// Adds a generic item at the back of the deque.
METHOD Enqueue_Generic : I_Deque
VAR_INPUT
	Item : T_Generic; // Item to store.
	bAt_Front : BOOL; // Enqueues at front if set to TRUE.
END_VAR
VAR_OUTPUT
	bSuccess : BOOL;
END_VAR
Enqueue_Generic := THIS^;

IF bAt_Front THEN
	THIS^.fbList.Insert_Generic(0, Item, bSuccess => bSuccess);
ELSE
	THIS^.fbList.Insert_Generic(THIS^.fbList._Count, Item, bSuccess => bSuccess);
	END_IF
END_METHOD

// Get item at the front of the deque without removing it.
METHOD Front : I_Deque
VAR_INPUT
	Item : ANY; // Variable to store returned item value
END_VAR
VAR_OUTPUT
	bSuccess : BOOL;
END_VAR
Front := THIS^;

THIS^.fbList.Get(0, Item, bSuccess => bSuccess);
END_METHOD

// Reverses the order of items in the deque.
METHOD Reverse : I_Deque
VAR_OUTPUT
	bSuccess : BOOL;
END_VAR
Reverse := THIS^;

THIS^.fbList.Reverse(bSuccess => bSuccess);
END_METHOD

END_FUNCTION_BLOCK

// POUs/Function Blocks/Collections/FB_List
// A doubly linked list with iterator hint optimisation.
// Essentially the linked list keeps track of the node it last accessed.
// Iteration starts from the closest node (head, tail or last accessed) to the access/mutation index.
// This should result in sequential access times of O(1) and similar times for access/mutation on the same index.
{attribute 'enable_dynamic_creation'}
{attribute 'no_assign'}
{attribute 'no_explicit_call' := 'direct call for this function block is not allowed'}
FUNCTION_BLOCK FB_List EXTENDS FB_Collection IMPLEMENTS I_List, I_Iterable//, I_Enumerable, I_Copyable
VAR
	pHead, pTail, pLast_Accessed : POINTER TO T_List_Node;
	Last_Accessed_Index : T_Position := -1;
END_VAR

// Iteration helper method that finds the closest node to an index and iterates from there to the node at the specified index.
METHOD PROTECTED Closest_Node_Iterator : POINTER TO T_List_Node
VAR_INPUT
	Index : T_Position;
END_VAR
VAR
	pTmp : POINTER TO T_List_Node;
	Dist, Last_Access_Dist,
	Head_Dist, Tail_Dist : T_Position;
END_VAR
Last_Access_Dist := ABS(THIS^.Last_Accessed_Index - Index);
Head_Dist := Index;
Tail_Dist := THIS^._Count - Index - 1;

Dist := MIN(Last_Access_Dist, Head_Dist, Tail_Dist);

Closest_Node_Iterator := THIS^.Iterate(
	SEL(Dist = Head_Dist, SEL(Dist = Tail_Dist,  THIS^.pLast_Accessed, THIS^.pTail), THIS^.pHead), // Select the closest node to start iteration.
	Dist, // get the smallest displacement
	SEL(Dist = Head_Dist, SEL(Dist = Tail_Dist, Index > THIS^.Last_Accessed_Index, FALSE), TRUE)); // Set the iteration direction.
END_METHOD

// Iteration helper method to iterate from a given node in a specific direction for a specified count.
METHOD PROTECTED Iterate : POINTER TO T_List_Node
VAR_INPUT
	pStart 		: POINTER TO T_List_Node;
	Count 		: T_Capacity;
	bIterateUp 	: BOOL;
END_VAR
VAR
	i : T_Capacity;
END_VAR
Iterate := pStart;
IF Count = 0 THEN RETURN; END_IF
IF bIterateUp THEN FOR i := 0 TO Count - 1 DO Iterate := Iterate^.pNext; END_FOR RETURN; END_IF
FOR i := 0 TO Count - 1 DO Iterate := Iterate^.pPrevious; END_FOR
END_METHOD

// Index of the first element.
PROPERTY _Begin : T_Position
GET
_Begin := 0;
END_GET
END_PROPERTY

// Index of the last element.
PROPERTY _End : T_Position
GET
_End := TO_DINT(THIS^._Count) - 1;
END_GET
END_PROPERTY

// Adds an item to the end of the list.
METHOD Append : I_List
VAR_INPUT
	Item : ANY; // Value to store in list
END_VAR
VAR_OUTPUT
	bSuccess : BOOL;
END_VAR
Append := THIS^;

THIS^.Insert_Generic(THIS^._Count, Item, bSuccess => bSuccess);
END_METHOD

// Empties/Clears/Deletes every item in the list.
METHOD Clear : I_List
VAR
	pTmp : POINTER TO T_List_Node;
END_VAR
Clear := THIS^;

WHILE THIS^.pHead <> 0 DO
	pTmp := THIS^.pHead^.pNext;
	F_Delete_Generic(THIS^.pHead^.Data);
	__DELETE(THIS^.pHead);
	THIS^.pHead := pTmp;
	END_WHILE

THIS^._Count := 0;	
THIS^.pTail := THIS^.pLast_Accessed := 0;
THIS^.Last_Accessed_Index := -1;
THIS^.Clear_Error();
END_METHOD

// Checks if item is contained in list.
METHOD Contains : BOOL
VAR_INPUT
	Item : ANY; // Item to find in list
END_VAR
THIS^.Search(Item, bSuccess => Contains);
END_METHOD

{attribute 'hide'}
METHOD FB_exit : BOOL
VAR_INPUT
	bInCopyCode : BOOL; // if TRUE, the exit method is called for exiting an instance that is copied afterwards (online change).
END_VAR
// If this is an online change or this collection is empty then ignore. 
IF bInCopyCode THEN RETURN; END_IF

THIS^.Clear();
END_METHOD

// Gets item from list at specified location without removing it
METHOD Get : I_List
VAR_INPUT
	Index : T_Position; // Location of item
	Item : ANY;  // Variable to store returned item
END_VAR
VAR_OUTPUT
	bSuccess : BOOL;
END_VAR
VAR
	Tmp : T_Generic;
END_VAR
Get := THIS^;

THIS^.Get_Generic(Index, Item => Tmp, bSuccess => bSuccess);

IF NOT bSuccess THEN RETURN; END_IF

IF NOT F_Matching_Generics(Item, Tmp) THEN
	THIS^._Error_Status := GVL_Errors.ERR_TYPE_MISMATCH;
	bSuccess := FALSE;
	RETURN;
	END_IF
	
F_Copy_Generic_Value(Tmp, Item, bSuccess => bSuccess, Error => THIS^.Error);
END_METHOD

// Returns item as a string, if type to string conversion is supported
METHOD Get_As_String : I_List
VAR_INPUT
	Index : T_Position; // Location of item
	sItem : REFERENCE TO STRING; // Variable to store returned item.
END_VAR
VAR_OUTPUT
	bSuccess : BOOL;
END_VAR
VAR
	Tmp : T_Generic;
END_VAR
Get_As_String := THIS^;

IF NOT __ISVALIDREF(sItem) THEN THIS^._Error_Status := GVL_Errors.ERR_INVALID_REFERENCE; RETURN; END_IF
	
THIS^.Get_Generic(Index, Item => Tmp, bSuccess => bSuccess);

IF NOT bSuccess THEN RETURN; END_IF
	
CASE Tmp.TypeClass OF
	T_Type.TYPE_STRING:
		Tc2_Utilities.STRNCPY(ADR(sItem), Tmp.pValue, MIN(Tc2_Utilities.LEN2(ADR(sItem))+1, TO_UDINT(Tmp.diSize)));
		THIS^.Clear_Error();

	T_Type.TYPE_WSTRING:
		Tc2_Utilities.WSTRING_TO_STRING2(ADR(sItem), Tmp.pValue, MIN(Tc2_Utilities.LEN2(ADR(sItem))+1, TO_UDINT(Tmp.diSize)));
		THIS^.Clear_Error();
ELSE
	sItem := F_Generic_To_String(Tmp, bSuccess => bSuccess, Error => THIS^.Error);
	END_CASE
END_METHOD

// Gets a value from a list in it's generic form.
// (** Use carefully as this contains the pointer of the actual value in the collection. **)
// If you wish to use this it is recommeded you create a copy of the returned value using MEMMOVE or MEMCPY
METHOD Get_Generic : I_List
VAR_INPUT
	Index : T_Position; // Location of item
END_VAR
VAR_OUTPUT
	Item : T_Generic := (TypeClass := T_Type.TYPE_NONE);
	bSuccess : BOOL;
END_VAR
VAR
	pTmp : POINTER TO T_List_Node;
END_VAR
Get_Generic := THIS^;

IF Index < 0 OR_ELSE Index >= THIS^._Count THEN
	// Throw out of bounds error.
	THIS^._Error_Status := GVL_Errors.ERR_INDEX_OUT_OF_BOUNDS;
	RETURN;
	END_IF
	
IF Index = 0 THEN
	Item := THIS^.pHead^.Data;
ELSIF Index = THIS^._Count - 1 THEN
	Item := THIS^.pTail^.Data;
ELSIF Index = THIS^.Last_Accessed_Index THEN
	Item := THIS^.pLast_Accessed^.Data;
ELSE
	pTmp := THIS^.Closest_Node_Iterator(Index);
	Item := pTmp^.Data;
	
	THIS^.Last_Accessed_Index := Index;
	THIS^.pLast_Accessed := pTmp;
	
	END_IF
	
bSuccess := TRUE;
THIS^.Clear_Error();
END_METHOD

// Gets the type of the item at specified location.
METHOD Get_Type_At : I_List
VAR_INPUT
	Index : T_Position;
END_VAR
VAR_OUTPUT
	Item_Type : T_Type := T_Type.TYPE_NONE;
	bSuccess : BOOL;
END_VAR
VAR
	Tmp : T_Generic;
END_VAR
Get_Type_At := THIS^;

THIS^.Get_Generic(Index, Item => Tmp, bSuccess => bSuccess);
Item_Type := Tmp.TypeClass;
END_METHOD

// Adds new item to list at specified location, if index = 0, item will be added at the front, if index = count, item will be added at the back
METHOD Insert : I_List
VAR_INPUT
	Index : T_Position; // Location of item
	Item : ANY; // Item to store in list
END_VAR
VAR_OUTPUT
	bSuccess : BOOL;
END_VAR
Insert := THIS^;

THIS^.Insert_Generic(Index, Item, bSuccess => bSuccess);
END_METHOD

// Adds new item to list at specified location using the generic form. 
// If index = 0, item will be added at the front, if index = count, item will be added at the back
METHOD Insert_Generic : I_List
VAR_INPUT
	Index 	 : T_Position; 	// Location of item
	Item 	 : T_Generic;  	// Item to store in list
END_VAR
VAR_OUTPUT
	bSuccess : BOOL;
END_VAR
VAR
	pTmp, pCurrent : POINTER TO ST_LIST_NODE;
END_VAR
Insert_Generic := THIS^;

IF Index < 0 OR_ELSE Index > THIS^._Count THEN
	// Throw out of bounds error.
	THIS^._Error_Status := GVL_Errors.ERR_INDEX_OUT_OF_BOUNDS;
	RETURN;
	END_IF
	
pTmp := __NEW(ST_LIST_NODE);
IF pTmp = 0 THEN THIS^._Error_Status := GVL_Errors.ERR_MALLOC_FAILED; RETURN; END_IF

pTmp^.Data := F_Clone_Generic(Item, bSuccess => bSuccess, Error => THIS^.Error);
IF NOT bSuccess THEN __DELETE(pTmp); RETURN; END_IF

IF Index = 0 THEN
	//...
	pTmp^.pNext := THIS^.pHead;
	IF THIS^.pHead <> 0 THEN THIS^.pHead^.pPrevious := pTmp; END_IF
	IF THIS^.pTail = 0 THEN THIS^.pTail := pTmp; END_IF
	THIS^.pHead := pTmp;
ELSIF Index = THIS^._Count THEN
	//...
	pTmp^.pPrevious := THIS^.pTail;
	IF THIS^.pTail <> 0 THEN THIS^.pTail^.pNext := pTmp; END_IF
	THIS^.pTail := pTmp;
ELSE	
	pCurrent := THIS^.Closest_Node_Iterator(Index);
	
	pTmp^.pNext := pCurrent;
	pTmp^.pPrevious := pCurrent^.pNext;
	pCurrent^.pPrevious^.pNext := pTmp;
	pCurrent^.pPrevious := pTmp;
	
	THIS^.Last_Accessed_Index := Index;
	THIS^.pLast_Accessed := pTmp;
	END_IF
	
THIS^.Increment_Count();
END_METHOD

// Adds an item at the front of the list.
METHOD Prepend : I_List
VAR_INPUT
	Item : ANY; // Value to store in list
END_VAR
VAR_OUTPUT
	bSuccess : BOOL;
END_VAR
Prepend := THIS^;

THIS^.Insert_Generic(0, Item, bSuccess => bSuccess);
END_METHOD

// Removes item from the list.
METHOD Remove : I_List
VAR_INPUT
	Item : ANY; // Item to remove from in list
END_VAR
VAR_OUTPUT
	bSuccess : BOOL;
END_VAR
VAR
	Tmp : T_Position;
END_VAR
Remove := THIS^;

THIS^.Search(Item, Index => Tmp, bSuccess => bSuccess);
IF NOT bSuccess THEN RETURN; END_IF 
THIS^.Remove_At(Tmp, bSuccess => bSuccess);
END_METHOD

// Remove item at specified location 
METHOD Remove_At : I_List
VAR_INPUT
	Index : T_Position; // Location of item
END_VAR
VAR_OUTPUT
	bSuccess : BOOL;
END_VAR
VAR
	pTmp : POINTER TO T_List_Node;
END_VAR
Remove_At := THIS^;

IF Index < 0 OR_ELSE Index >= THIS^._Count THEN
	// Throw out of bounds error.
	THIS^._Error_Status := GVL_Errors.ERR_INDEX_OUT_OF_BOUNDS;
	RETURN;
	END_IF

IF Index = 0 THEN
	//...
	pTmp := THIS^.pHead;
	IF THIS^.pHead = THIS^.pTail THEN
		THIS^.pLast_Accessed := THIS^.pTail := 0;
		THIS^.Last_Accessed_Index := -1;
		END_IF
		
	THIS^.pHead := THIS^.pHead^.pNext;
	
	F_Delete_Generic(pTmp^.Data);
	__DELETE(pTmp);
	
ELSIF Index = THIS^._Count - 1 THEN
	//...
	pTmp := THIS^.pTail^.pPrevious;
	THIS^.pTail := pTmp;
	F_Delete_Generic(pTmp^.pNext^.Data);
	__DELETE(pTmp^.pNext);
ELSE
	//...	
	pTmp := THIS^.Closest_Node_Iterator(Index);
	
	// Do deletion
	pTmp^.pNext^.pPrevious := pTmp^.pPrevious;
	pTmp^.pPrevious^.pNext := pTmp^.pNext;
	
	THIS^.Last_Accessed_Index := -1;
	THIS^.pLast_Accessed := 0;
	
	THIS^.Last_Accessed_Index := Index;
	THIS^.pLast_Accessed := pTmp^.pNext;
	
	F_Delete_Generic(pTmp^.Data);
	__DELETE(pTmp);
	END_IF
	
THIS^.Decrement_Count();
bSuccess := TRUE;
THIS^.Clear_Error();
END_METHOD

// Removes item at the back of the list.
METHOD Remove_Last : I_List
VAR_OUTPUT
	bSuccess : BOOL;
END_VAR
Remove_Last := THIS^.Remove_At(THIS^._Count - 1, bSuccess => bSuccess);
END_METHOD

// Manually resize list. If list becomes smaller, item on higher locations will be deleted.
METHOD Resize : I_List
VAR_INPUT
	Size : T_Capacity; // New size of list.
END_VAR
VAR_OUTPUT
	bSuccess : BOOL;
END_VAR
VAR
	Tmp : T_Generic := (TypeClass := T_Type.TYPE_NONE);
END_VAR
Resize := THIS^;

IF Size = 0 THEN 
	THIS^.Clear();
ELSE
	WHILE THIS^._Count > Size DO 
		THIS^.Remove_At(THIS^._Count - 1, bSuccess => bSuccess);
		IF NOT bSuccess THEN RETURN; END_IF 
		END_WHILE
	WHILE THIS^._Count < Size DO 
		THIS^.Insert_Generic(THIS^._Count, Tmp, bSuccess => bSuccess);
		IF NOT bSuccess THEN RETURN; END_IF 
		END_WHILE
	END_IF
END_METHOD

// Reverses the order of items in the list
METHOD Reverse : I_List
VAR_OUTPUT
	bSuccess : BOOL;
END_VAR
VAR
	pFront, pBack : POINTER TO T_List_Node;
END_VAR
Reverse := THIS^;

IF THIS^._Empty THEN bSuccess := TRUE; THIS^.Clear_Error(); RETURN; END_IF

pFront := THIS^.pHead;
pBack := THIS^.pTail;

WHILE (pFront <> pBack) AND_THEN (pFront^.pPrevious <> pBack) DO
	F_Swap_Generics(pFront^.Data, pBack^.Data);
	pFront := pFront^.pNext;
	pBack := pBack^.pPrevious;
	END_WHILE
	
bSuccess := TRUE;
THIS^.Clear_Error();
END_METHOD

// Find the location of an item in list.
METHOD Search : I_List
VAR_INPUT
	Item : ANY; // Item to find in list
END_VAR
VAR_OUTPUT
	Index : T_Position := -1; //Location of item in list 
	bSuccess : BOOL;
END_VAR
VAR
	i : T_Position;
	pTmp : POINTER TO T_List_Node;
END_VAR
Search := THIS^;

pTmp := THIS^.pHead; 
WHILE pTmp <> 0 DO
	CASE F_Compare_Generics(Item, pTmp^.Data) OF
		T_Comparison.Equal:
			bSuccess := TRUE;
			THIS^.Clear_Error();
			Index := i;
			RETURN;
		END_CASE
	pTmp := pTmp^.pNext;	
	i := i + 1;
	END_WHILE

// Throw item not found error.
THIS^._Error_Status := GVL_Errors.ERR_NO_ITEM;
END_METHOD

// Changes the item at the specified location in the list.
METHOD Set : I_List
VAR_INPUT
	Index 	: T_Position; // Location of item
	Item 	: ANY; 	// Item to store in list
END_VAR
VAR_OUTPUT
	bSuccess : BOOL;
END_VAR
Set := THIS^;

THIS^.Set_Generic(Index, Item, bSuccess => bSuccess);
END_METHOD

// Changes the item at the specified location in the list in it's generic form.
METHOD Set_Generic : I_List
VAR_INPUT
	Index : T_Position; // Location of item
	Item : T_Generic; // Item to store in list
END_VAR
VAR_OUTPUT
	bSuccess : BOOL;
END_VAR
VAR
	pTmp : POINTER TO T_List_Node;
	Tmp : T_Generic;
END_VAR
Set_Generic := THIS^;

IF Index < 0 OR_ELSE Index >= THIS^._Count THEN
	// Throw out of bounds error.
	THIS^._Error_Status := GVL_Errors.ERR_INDEX_OUT_OF_BOUNDS;
	RETURN;
	END_IF
	
IF Index = 0 THEN
	Tmp := F_Clone_Generic(Item, bSuccess => bSuccess, Error => THIS^.Error);
	IF NOT bSuccess THEN RETURN; END_IF
	F_Delete_Generic(THIS^.pHead^.Data);
	THIS^.pHead^.Data := Tmp;
	
ELSIF Index = THIS^._Count - 1 THEN
	Tmp := F_Clone_Generic(Item, bSuccess => bSuccess, Error => THIS^.Error);
	IF NOT bSuccess THEN RETURN; END_IF
	F_Delete_Generic(THIS^.pTail^.Data);
	THIS^.pTail^.Data := Tmp;
	
ELSIF Index = THIS^.Last_Accessed_Index THEN
	Tmp := F_Clone_Generic(Item, bSuccess => bSuccess, Error => THIS^.Error);
	IF NOT bSuccess THEN RETURN; END_IF
	F_Delete_Generic(THIS^.pLast_Accessed^.Data);
	THIS^.pLast_Accessed^.Data := Tmp;
	 
ELSE
	Tmp := F_Clone_Generic(Item, bSuccess => bSuccess, Error => THIS^.Error);
	IF NOT bSuccess THEN RETURN; END_IF
	pTmp := THIS^.Closest_Node_Iterator(Index);
	F_Delete_Generic(pTmp^.Data);
	pTmp^.Data := Tmp;

	THIS^.Last_Accessed_Index := Index;
	THIS^.pLast_Accessed := pTmp;
	END_IF
END_METHOD

// Swaps item at index A with item at index B.
METHOD Swap : I_List
VAR_INPUT
	Index_A, Index_B : T_Position;
END_VAR
VAR_OUTPUT
	bSuccess : BOOL;
END_VAR
Swap := THIS^;

IF Index_A < 0 OR_ELSE Index_A >= THIS^._Count OR_ELSE Index_B < 0 OR_ELSE Index_B >= THIS^._Count THEN
	THIS^._Error_Status := GVL_Errors.ERR_INDEX_OUT_OF_BOUNDS;
	RETURN;
	END_IF
	
F_Swap_Generics(THIS^.Closest_Node_Iterator(Index_A)^.Data, THIS^.Closest_Node_Iterator(Index_B)^.Data, bSuccess => bSuccess, Error => THIS^.Error);
END_METHOD

END_FUNCTION_BLOCK

// POUs/Function Blocks/Collections/FB_Hash_Map
// A collection of key value pairs items.
// Implemented using hash table with closed addressing.
{attribute 'enable_dynamic_creation'}
{attribute 'no_assign'}
{attribute 'no_explicit_call' := 'direct call for this function block is not allowed'}
FUNCTION_BLOCK FB_Hash_Map EXTENDS FB_Collection IMPLEMENTS I_Hash_Map
VAR
	pBuckets : POINTER TO POINTER TO T_Hashmap_Bucket_Node; // Array of pointers to hash bucket node.
	Bucket_Count : T_Capacity;
	pKeys, pValues : POINTER TO FB_Array_List;
	fbImmutable_Keys_List,
	fbImmutable_Values_List : FB_Immutable_List;
	bKeys_Updated, bValues_Updated : BOOL := TRUE;
END_VAR
VAR CONSTANT
	fLoad_Factor : REAL := 0.75;
END_VAR

// Creates buckets and initialises them since user defined types can't be created as arrays dynamically using __NEW(...).
METHOD PROTECTED Create_Buckets : POINTER TO POINTER TO T_Hashmap_Bucket_Node
VAR_INPUT
	Count : T_Capacity;
END_VAR
VAR_OUTPUT
	bSuccess : BOOL := TRUE;
	Error : T_Error := GVL_Errors.ERR_NO_ERROR;
END_VAR
VAR
	i : T_Capacity;
END_VAR
IF Count <= 0 THEN RETURN; END_IF

Create_Buckets := __NEW(POINTER TO ST_HASHMAP_BUCKET_NODE, TO_UDINT(Count));

IF Create_Buckets = 0 THEN
	bSuccess := FALSE;
	Error := GVL_Errors.ERR_MALLOC_FAILED;
	END_IF
END_METHOD

// Creates a new node in dynamic memory with a clone of the generic item as it data.
METHOD PROTECTED Create_Node : POINTER TO ST_HASHMAP_BUCKET_NODE
VAR_INPUT
	Key, Value : T_Generic;
END_VAR
VAR_OUTPUT
	bSuccess : BOOL;
	Error : T_Error;
END_VAR
Create_Node := __NEW(ST_HASHMAP_BUCKET_NODE);

IF Create_Node = 0 THEN 
	Error := GVL_Errors.ERR_MALLOC_FAILED;
	RETURN;
	END_IF

Create_Node^.Key := F_Clone_Generic(Key, bSuccess => bSuccess, Error => Error);

IF NOT bSuccess THEN __DELETE(Create_Node); RETURN; END_IF

Create_Node^.Value := F_Clone_Generic(Value, bSuccess => bSuccess, Error => Error);

IF NOT bSuccess THEN
	F_Delete_Generic(Create_Node^.Key);
	__DELETE(Create_Node);
	END_IF
END_METHOD

// Safety deletes node.
// If the node and/or it's value/data is in dynamic memory it/they will be deleted.
METHOD PROTECTED Delete_Node
VAR_INPUT
	pNode : REFERENCE TO POINTER TO T_Hashmap_Bucket_Node;
END_VAR
IF (pNode = 0) THEN RETURN; END_IF 

F_Delete_Generic(pNode^.Key);
F_Delete_Generic(pNode^.Value);

CASE Tc2_System.F_CheckMemoryArea(pNode, 1) OF
	Tc2_System.E_TcMemoryArea.Dynamic: __DELETE(pNode);
ELSE
	pNode := 0;
	END_CASE
END_METHOD

// Wrapper for murmur3 hash function that generates a value that fits in the upperage of DINT to avoid negative values due to integer overflow.
METHOD PROTECTED Hash : T_Capacity
VAR_INPUT
	Data : T_Generic;
END_VAR
Hash := TO_DINT(F_Murmur3_Hash(Data) MOD TO_DWORD(GVL_Constants.MAX_CAPACITY));
END_METHOD

// Number of buckets in the hash map.
PROPERTY _Bucket_Count : T_Capacity;
GET
_Bucket_Count := THIS^.Bucket_Count;
END_GET
SET
PROTECTED 
VAR
END_VAR
THIS^.Bucket_Count := _Bucket_Count;
END_SET
END_PROPERTY

// Empties/Clears/Deletes every item in the map.
METHOD Clear : I_Map
VAR
	i : T_Capacity;
	pCurrent, pNext : POINTER TO T_Hashmap_Bucket_Node;
END_VAR
Clear := THIS^;

FOR i := 0 TO THIS^._Bucket_Count - 1 DO
	pCurrent := THIS^.pBuckets[i];
	WHILE pCurrent <> 0 DO
		pNext := pCurrent^.pNext;
		THIS^.Delete_Node(pCurrent);
		pCurrent := pNext;
		END_WHILE
	END_FOR

IF THIS^.pKeys <> 0 THEN
	THIS^.fbImmutable_Keys_List(ipList := 0);  
	__DELETE(THIS^.pKeys); 
	END_IF
	
IF THIS^.pValues <> 0 THEN 
	THIS^.fbImmutable_Values_List(ipList := 0);
	__DELETE(THIS^.pValues);
	END_IF

__DELETE(THIS^.pBuckets);
THIS^._Bucket_Count := 0;
THIS^._Count := 0;
THIS^.bKeys_Updated := THIS^.bValues_Updated := TRUE;
END_METHOD

// Checks if key is contained in the map.
METHOD Contains : BOOL
VAR_INPUT
	Key : ANY; // Key to find.
END_VAR
VAR
	Index : T_Position;
	pCurrent : POINTER TO T_Hashmap_Bucket_Node;
END_VAR
IF THIS^._Empty THEN RETURN; END_IF

Index := THIS^.Hash(Key) MOD THIS^.Bucket_Count;

pCurrent := THIS^.pBuckets[Index];

WHILE pCurrent <> 0 DO
	IF F_Compare_Generics(Key, pCurrent^.Key) = T_Comparison.Equal THEN 
		Contains := TRUE;
		THIS^.Clear_Error();
		RETURN; 
		END_IF
	pCurrent := pCurrent^.pNext;
	END_WHILE
END_METHOD

{attribute 'hide'}
METHOD FB_exit : BOOL
VAR_INPUT
	bInCopyCode : BOOL; // if TRUE, the exit method is called for exiting an instance that is copied afterwards (online change).
END_VAR
// Return if it's an online change.
IF bInCopyCode THEN RETURN; END_IF

THIS^.Clear();
END_METHOD

{attribute 'hide'}
METHOD FB_init : BOOL
VAR_INPUT
	bInitRetains : BOOL; // if TRUE, the retain variables are initialized (warm start / cold start)
	bInCopyCode : BOOL;  // if TRUE, the instance afterwards gets moved into the copy code (online change)
	Initial_Bucket_Count : T_Capacity; // Number of buckets you want to initialise the hash map with. Use 0 if you don't know.
END_VAR
VAR 
	bSuccess : BOOL;
END_VAR
// Return if it's an online change.
IF bInCopyCode THEN RETURN; END_IF

THIS^.pBuckets := THIS^.Create_Buckets(Initial_Bucket_Count, bSuccess => bSuccess, Error => THIS^.Error);
THIS^._Bucket_Count := SEL(THIS^.pBuckets <> 0, 0,Initial_Bucket_Count);
END_METHOD

// Gets the value associated with the specified key without removing it from the map.
METHOD Get : I_Map
VAR_INPUT
	Key : ANY; // Key used to identify stored value
	Value : ANY; // Variable to store requested data 
END_VAR
VAR_OUTPUT
	bSuccess : BOOL;
END_VAR
VAR
	Tmp : T_Generic;
END_VAR
Get := THIS^;

THIS^.Get_Generic(Key, Value => Tmp, bSuccess => bSuccess);

IF NOT bSuccess THEN RETURN; END_IF

IF NOT F_Matching_Generics(Value, Tmp) THEN
	THIS^._Error_Status := GVL_Errors.ERR_TYPE_MISMATCH;
	RETURN;
	END_IF
	
F_Copy_Generic_Value(Tmp, Value, bSuccess => bSuccess, Error => THIS^.Error);
END_METHOD

// Returns value as a string, if type to string conversion is supported.
METHOD Get_As_String : I_Map
VAR_INPUT
	Key : ANY; // Key used to identify stored value
	sValue : REFERENCE TO STRING; // Variable to store returned item.
END_VAR
VAR_OUTPUT
	bSuccess : BOOL;
END_VAR
VAR
	Tmp : T_Generic;
END_VAR
Get_As_String := THIS^;

IF NOT __ISVALIDREF(sValue) THEN 
	THIS^._Error_Status := GVL_Errors.ERR_INVALID_REFERENCE;
	RETURN;
	END_IF
	
THIS^.Get_Generic(Key, Value => Tmp, bSuccess => bSuccess);

IF NOT bSuccess THEN RETURN; END_IF
	
CASE Tmp.TypeClass OF
	T_Type.TYPE_STRING:
		Tc2_Utilities.STRNCPY(ADR(sValue), Tmp.pValue, MIN(Tc2_Utilities.LEN2(ADR(sValue))+1, TO_UDINT(Tmp.diSize)));
		THIS^.Clear_Error();

	T_Type.TYPE_WSTRING:
		Tc2_Utilities.WSTRING_TO_STRING2(ADR(sValue), Tmp.pValue, MIN(Tc2_Utilities.LEN2(ADR(sValue))+1, TO_UDINT(Tmp.diSize)));
		THIS^.Clear_Error();
ELSE
	sValue := F_Generic_To_String(Tmp, bSuccess => bSuccess, Error => THIS^.Error);
	END_CASE
END_METHOD

// Gets the value in its generic form associated with the specified key in its generic form without removing it from the map.
// (** Use carefully as this contains the pointer of the actual value in the collection. **)
// If you wish to use this it is recommeded you create a copy of the returned value using MEMCPY
METHOD Get_Generic : I_Map
VAR_INPUT
	Key : T_Generic; // Key used to identify stored value
END_VAR
VAR_OUTPUT
	Value : T_Generic; // Variable to store requested data 
	bSuccess : BOOL;
END_VAR
VAR
	Index : T_Position;
	pCurrent : POINTER TO T_Hashmap_Bucket_Node;
END_VAR
Get_Generic := THIS^;

IF THIS^._Empty THEN THIS^._Error_Status := GVL_Errors.ERR_NO_KEY; RETURN; END_IF

Index := THIS^.Hash(Key) MOD THIS^.Bucket_Count;

pCurrent := THIS^.pBuckets[Index];

WHILE pCurrent <> 0 DO
	IF F_Compare_Generics(Key, pCurrent^.Key) = T_Comparison.Equal THEN
		Value := pCurrent^.Value;
		bSuccess := TRUE;
		THIS^.Clear_Error();
		RETURN; 
		END_IF
	pCurrent := pCurrent^.pNext;
	END_WHILE
	
THIS^._Error_Status := GVL_Errors.ERR_NO_KEY;
END_METHOD

// Gets an immutable list of the keys.
METHOD Get_Keys : I_Immutable_List
VAR
	i : T_Capacity;
	pCurrent : POINTER TO T_Hashmap_Bucket_Node;
END_VAR
IF THIS^.pKeys = 0 THEN THIS^.pKeys := __NEW(FB_Array_List(Initial_Capacity := 0)); END_IF
THIS^.fbImmutable_Keys_List(ipList := THIS^.pKeys^);
Get_Keys := THIS^.fbImmutable_Keys_List;

IF NOT THIS^.bKeys_Updated THEN RETURN; END_IF

THIS^.pKeys^.Clear();

IF THIS^._Empty THEN RETURN; END_IF

FOR i := 0 TO THIS^._Bucket_Count - 1 DO
	pCurrent := THIS^.pBuckets[i];
	WHILE pCurrent <> 0 DO
		pKeys^.Insert_Generic(pKeys^._Count, pCurrent^.Key);
		pCurrent := pCurrent^.pNext;
		END_WHILE
	END_FOR
	
THIS^.bKeys_Updated := FALSE;
END_METHOD

// Gets an immutable list of the values.
METHOD Get_Values : I_Immutable_List
VAR
	i : T_Capacity;
	pCurrent : POINTER TO T_Hashmap_Bucket_Node;
END_VAR
IF THIS^.pValues = 0 THEN THIS^.pValues := __NEW(FB_Array_List(Initial_Capacity := 0)); END_IF
THIS^.fbImmutable_Values_List(ipList := THIS^.pValues^);
Get_Values := THIS^.fbImmutable_Values_List;

IF NOT THIS^.bValues_Updated THEN RETURN; END_IF

pValues^.Clear();

IF THIS^._Empty THEN RETURN; END_IF

FOR i := 0 TO THIS^._Bucket_Count - 1 DO
	pCurrent := THIS^.pBuckets[i];
	WHILE pCurrent <> 0 DO
		pValues^.Insert_Generic(pValues^._Count, pCurrent^.Value);
		pCurrent := pCurrent^.pNext;
		END_WHILE
	END_FOR
	
THIS^.bValues_Updated := FALSE;
END_METHOD

// Insert an element with the provided key and value to the map.
METHOD Insert : I_Map
VAR_INPUT
	Key : ANY; // Key used to identify stored value
	Value : ANY; // Value to store in map with key
END_VAR
VAR_OUTPUT
	bSuccess : BOOL;
END_VAR
Insert := THIS^.Insert_Generic(Key, Value, FALSE, bSuccess => bSuccess);
END_METHOD

// Insert an element with the provided key and value in their generic forms to the map.
METHOD Insert_Generic : I_Map
VAR_INPUT
	Key : T_Generic; // Key used to identify stored value
	Value : T_Generic; // Value to store in map with key
	bUpdate : BOOL; // If this is true the value will be updated if the key already exists.
END_VAR
VAR_OUTPUT
	bSuccess : BOOL;
END_VAR
VAR
	Index : T_Position;
	pCurrent : POINTER TO T_Hashmap_Bucket_Node;
	Tmp : T_Generic;
END_VAR
Insert_Generic := THIS^;

IF TO_REAL(THIS^._Count) > (TO_REAL(THIS^._Bucket_Count) * THIS^.fLoad_Factor) OR_ELSE THIS^.Bucket_Count <= 0 THEN
	// Increasing the bucket by 50% once the load factor is reached.
	// Bitwise shifting is the same as multiplying by 1.5, this is done because no complicated casting is needed.
	THIS^.Resize(SEL(THIS^._Bucket_Count > 1, 16, THIS^._Bucket_Count + SHR(THIS^._Bucket_Count, 1)), bSuccess => bSuccess);
	IF NOT bSuccess THEN RETURN; END_IF
	END_IF

Index := THIS^.Hash(Key) MOD THIS^._Bucket_Count;

pCurrent := THIS^.pBuckets[Index];

WHILE pCurrent <> 0 DO
	CASE F_Compare_Generics(Key, pCurrent^.Key) OF
		T_Comparison.Equal:
			IF bUpdate THEN
				Tmp := F_Clone_Generic(Value, bSuccess => bSuccess, Error => THIS^.Error);
				IF NOT bSuccess THEN RETURN; END_IF
				F_Delete_Generic(pCurrent^.Value);
				pCurrent^.Value := Tmp;
				THIS^.bValues_Updated := TRUE;
			ELSE
				THIS^._Error_Status := GVL_Errors.ERR_DUPLICATE_KEY;
			END_IF
			RETURN;
		T_Comparison.Invalid:
			THIS^._Error_Status := GVL_Errors.ERR_INVALID_COMPARISON;
			RETURN;
	ELSE
		pCurrent := pCurrent^.pNext; 
		END_CASE
	END_WHILE
	
pCurrent := THIS^.Create_Node(Key, Value, bSuccess => bSuccess, Error => THIS^.Error);
IF NOT bSuccess THEN RETURN; END_IF
pCurrent^.pNext := THIS^.pBuckets[Index];
THIS^.pBuckets[Index] := pCurrent;

THIS^.Increment_Count();
THIS^.bKeys_Updated := THIS^.bValues_Updated := TRUE;
END_METHOD

// Removes value with the specified key from the map.
METHOD Remove : I_Map
VAR_INPUT
	Key : ANY; // Key used to identify stored value
END_VAR
VAR_OUTPUT
	bSuccess : BOOL;
END_VAR
Remove := THIS^.Remove_Generic(Key, bSuccess => bSuccess);
END_METHOD

// Removes value with the specified key in its generic form from the map.
METHOD Remove_Generic : I_Map
VAR_INPUT
	Key : T_Generic; // Key used to identify stored value
END_VAR
VAR_OUTPUT
	bSuccess : BOOL;
END_VAR
VAR
	Index : T_Position;
	pCurrent, pPrevious : POINTER TO T_Hashmap_Bucket_Node;
END_VAR
Remove_Generic := THIS^;

IF THIS^._Empty THEN THIS^._Error_Status := GVL_Errors.ERR_NO_KEY; RETURN; END_IF

Index := THIS^.Hash(Key) MOD THIS^.Bucket_Count;

pCurrent := THIS^.pBuckets[Index];

WHILE pCurrent <> 0 DO
	IF F_Compare_Generics(Key, pCurrent^.Key) = T_Comparison.Equal THEN
		IF pPrevious <> 0 THEN 
			pPrevious^.pNext := pCurrent^.pNext;
		ELSE
			THIS^.pBuckets[Index] := pCurrent^.pNext;
			END_IF
		THIS^.Delete_Node(pCurrent);
		bSuccess := TRUE;
		THIS^.Decrement_Count();
		THIS^.bKeys_Updated := THIS^.bValues_Updated := TRUE;
		THIS^.Clear_Error();
		RETURN;
		END_IF
		
	pPrevious := pCurrent;
	pCurrent := pCurrent^.pNext;
	END_WHILE
	
THIS^._Error_Status := GVL_Errors.ERR_NO_KEY;
END_METHOD

// Sets the number of buckets in the hash map.
// Existing items are rehashed and redistributed into the new buckets.
// Note that of the count is 0 the hashtable is cleared.
METHOD Resize : I_Hash_Map
VAR_INPUT
	Count : T_Capacity;
END_VAR
VAR_OUTPUT
	bSuccess : BOOL;
END_VAR
VAR
	Hash : DWORD;
	New_Index : T_Position;
	i : T_Capacity;
	pCurrent, pNext : POINTER TO T_Hashmap_Bucket_Node;
	pNew_Bucket : POINTER TO POINTER TO T_Hashmap_Bucket_Node;
END_VAR
Resize := THIS^;

IF Count < 0 THEN THIS^._Error_Status := GVL_Errors.ERR_INDEX_OUT_OF_BOUNDS; RETURN; END_IF
IF Count = 0 THEN THIS^.Clear(); bSuccess := TRUE; THIS^.Clear_Error(); RETURN; END_IF
IF Count = THIS^._Bucket_Count THEN bSuccess := TRUE; THIS^.Clear_Error(); RETURN; END_IF

pNew_Bucket := THIS^.Create_Buckets(Count, bSuccess => bSuccess, Error => THIS^.Error);

IF NOT bSuccess THEN RETURN; END_IF;

FOR i := 0 TO THIS^._Bucket_Count - 1 DO
	pCurrent := THIS^.pBuckets[i];
	WHILE pCurrent <> 0 DO
		pNext := pCurrent^.pNext;
		New_Index := THIS^.Hash(pCurrent^.Key) MOD Count;
		pCurrent^.pNext := pNew_Bucket[New_Index];
		pNew_Bucket[New_Index] := pCurrent;
		pCurrent := pNext;
		END_WHILE
	END_FOR
	
__DELETE(THIS^.pBuckets);
THIS^.pBuckets := pNew_Bucket;
THIS^._Bucket_Count := Count;
END_METHOD

// Updates the value at the provided key with the new value in the map.
METHOD Update : I_Map
VAR_INPUT
	Key 	: ANY; // Key used to identify stored value
	Value 	: ANY; // Value to store in map with key
END_VAR
VAR_OUTPUT
	bSuccess : BOOL;
END_VAR
Update := THIS^.Update_Generic(Key, Value, bSuccess => bSuccess);
END_METHOD

// Updates the value at the provided key with the new value in their generic forms in the map.
METHOD Update_Generic : I_Map
VAR_INPUT
	Key 	: T_Generic; // Key used to identify stored value
	Value 	: T_Generic; // Value to store in map with key
END_VAR
VAR_OUTPUT
	bSuccess : BOOL;
END_VAR
VAR
	Index : T_Position;
	pCurrent : POINTER TO T_Hashmap_Bucket_Node;
	Tmp : T_Generic;
END_VAR
Update_Generic := THIS^;

IF THIS^._Empty THEN THIS^._Error_Status := GVL_Errors.ERR_NO_KEY; RETURN; END_IF

Index := THIS^.Hash(Key) MOD THIS^.Bucket_Count;

pCurrent := THIS^.pBuckets[Index];

WHILE pCurrent <> 0 DO
	CASE F_Compare_Generics(Key, pCurrent^.Key) OF
		T_Comparison.Equal:
			Tmp := F_Clone_Generic(Value, bSuccess => bSuccess, Error => THIS^.Error);
			IF NOT bSuccess THEN RETURN; END_IF;
			F_Delete_Generic(pCurrent^.Value);
			pCurrent^.Value := Tmp;
			THIS^.bValues_Updated := TRUE;
			RETURN;
		T_Comparison.Invalid:
			THIS^._Error_Status := GVL_Errors.ERR_INVALID_COMPARISON;
			RETURN;
	ELSE
		pCurrent := pCurrent^.pNext; 
		END_CASE
	END_WHILE
	
THIS^._Error_Status := GVL_Errors.ERR_NO_KEY;
END_METHOD

// Updates a value in the map for a given key. If the key doesnt exist, it will be inserted.
METHOD Upsert : I_Map
VAR_INPUT
	Key 	: ANY; // Key used to identify stored value
	Value 	: ANY; // Value to store in map with key
END_VAR
VAR_OUTPUT
	bSuccess : BOOL;
END_VAR
Upsert := THIS^.Insert_Generic(Key, Value, TRUE, bSuccess => bSuccess);
END_METHOD

END_FUNCTION_BLOCK

// POUs/Functions/F_Murmur3_Hash
// Generates a 32-bit hash code using MurmurHash3, created by Austin Appleby. Source: https://en.wikipedia.org/wiki/MurmurHash
FUNCTION F_Murmur3_Hash : DWORD
VAR_INPUT
	Data : T_Generic;
END_VAR
VAR
	i, nSize 	: UDINT;
	nK, nHash 	: DWORD;
END_VAR

CASE Data.TypeClass OF
	__SYSTEM.TYPE_CLASS.TYPE_STRING:
		nSize := Tc2_Utilities.LEN2(Data.pValue);
	__SYSTEM.TYPE_CLASS.TYPE_WSTRING:
		nSize := Tc2_Utilities.WLEN2(Data.pValue)*2;
ELSE
		nSize := TO_UDINT(Data.diSize);
END_CASE

FOR i := SHR(nSize, 2) TO 1 BY -1 DO
	MEMCPY(ADR(nK), Data.pValue, SIZEOF(DWORD));
	Data.pValue := Data.pValue + SIZEOF(DWORD);
	nHash := nHash XOR F_Murmur_Scramble(nK);
	nHash := SHL(nHash,13) OR SHR(nHash,19);
	nHash := nHash * 5 + 16#E6546B64;
	END_FOR
	
nK := 0;
FOR i := (nSize AND 3) TO 1 BY -1 DO
	nK := SHL(nK,8);
	nK := nK OR Data.pValue[i-1];
	END_FOR

nHash := nHash XOR F_Murmur_Scramble(nK);
nHash := nHash XOR nSize;
nHash := nHash XOR SHR(nHash, 16);
nHash := nHash * 16#85EBCA6B;
nHash := nHash XOR SHR(nHash, 13);
nHash := nHash * 16#C2B2AE35;
nHash := nHash XOR SHR(nHash, 16); 

F_Murmur3_Hash := nHash;

END_FUNCTION

// POUs/Functions/F_Murmur_Scramble
FUNCTION INTERNAL F_Murmur_Scramble : DWORD
VAR_INPUT
	nK : DWORD;
END_VAR
VAR
END_VAR

nK := nK * 16#CC9E2D51;
nK := SHL(nK, 15) OR SHR(nK, 17);
nK := nK * 16#1B873593;
F_Murmur_Scramble := nK;

END_FUNCTION

// POUs/Function Blocks/Collections/FB_Hash_Set
// A collection that contains no duplicate items.
// Implemented using hash table with closed addressing.
{attribute 'enable_dynamic_creation'}
{attribute 'no_assign'}
{attribute 'no_explicit_call' := 'direct call for this function block is not allowed'}
FUNCTION_BLOCK FB_Hash_Set EXTENDS FB_Collection IMPLEMENTS I_Hash_Set
VAR
	pBuckets : POINTER TO POINTER TO T_Hashset_Bucket_Node; // Array of pointers to hash bucket node.
	Bucket_Count : T_Capacity;
	pValues : POINTER TO FB_Array_List;
	fbImmutable_Values_List : FB_Immutable_List;
	bValues_Updated : BOOL := TRUE;
END_VAR
VAR CONSTANT
	fLoad_Factor : REAL := 0.75;
END_VAR

// Creates buckets and initialises them since user defined types can't be created as arrays dynamically using __NEW(...).
METHOD PROTECTED Create_Buckets : POINTER TO POINTER TO T_Hashset_Bucket_Node
VAR_INPUT
	Count : T_Capacity;
END_VAR
VAR_OUTPUT
	bSuccess : BOOL := TRUE;
	Error : T_Error := GVL_Errors.ERR_NO_ERROR;
END_VAR
VAR
	i : T_Capacity;
END_VAR
IF Count <= 0 THEN RETURN; END_IF

Create_Buckets := __NEW(POINTER TO ST_HASHSET_BUCKET_NODE, TO_UDINT(Count));

IF Create_Buckets = 0 THEN
	bSuccess := FALSE;
	Error := GVL_Errors.ERR_MALLOC_FAILED;
	END_IF
END_METHOD

// Creates a new node in dynamic memory with a clone of the generic item as it data.
METHOD PROTECTED Create_Node : POINTER TO ST_HASHSET_BUCKET_NODE
VAR_INPUT
	Item : T_Generic;
END_VAR
VAR_OUTPUT
	bSuccess : BOOL;
	Error : T_Error;
END_VAR
Create_Node := __NEW(ST_HASHSET_BUCKET_NODE);

IF Create_Node = 0 THEN 
	Error := GVL_Errors.ERR_MALLOC_FAILED;
	RETURN;
	END_IF

Create_Node^.Data := F_Clone_Generic(Item, bSuccess => bSuccess, Error => THIS^.Error);

IF NOT bSuccess THEN __DELETE(Create_Node); END_IF
END_METHOD

// Safety deletes node.
// If the node and/or it's value/data is in dynamic memory it/they will be deleted.
METHOD PROTECTED Delete_Node
VAR_INPUT
	pNode : REFERENCE TO POINTER TO T_Hashset_Bucket_Node;
END_VAR
IF (pNode = 0) THEN RETURN; END_IF 

F_Delete_Generic(pNode^.Data);

CASE Tc2_System.F_CheckMemoryArea(pNode, 1) OF
	Tc2_System.E_TcMemoryArea.Dynamic: __DELETE(pNode);
ELSE
	pNode := 0;
	END_CASE
END_METHOD

// Wrapper for murmur3 hash function that generates a value that fits in the upperage of DINT to avoid negative values due to integer overflow.
METHOD PROTECTED Hash : T_Capacity
VAR_INPUT
	Data : T_Generic;
END_VAR
Hash := TO_DINT(F_Murmur3_Hash(Data) MOD TO_DWORD(GVL_Constants.MAX_CAPACITY));
END_METHOD

// Number of buckets in the hash set.
PROPERTY _Bucket_Count : T_Capacity;
GET
_Bucket_Count := THIS^.Bucket_Count;
END_GET
SET
PROTECTED 
VAR
END_VAR
THIS^.Bucket_Count := _Bucket_Count;
END_SET
END_PROPERTY

// Empties/Clears/Deletes every item in the set.
METHOD Clear : I_Set
VAR
	i : T_Capacity;
	pCurrent, pNext : POINTER TO T_Hashset_Bucket_Node;
END_VAR
Clear := THIS^;

FOR i := 0 TO THIS^._Bucket_Count - 1 DO
	pCurrent := THIS^.pBuckets[i];
	WHILE pCurrent <> 0 DO
		pNext := pCurrent^.pNext;
		THIS^.Delete_Node(pCurrent);
		pCurrent := pNext;
		END_WHILE
	END_FOR

IF THIS^.pValues <> 0 THEN 
	THIS^.fbImmutable_Values_List(ipList := 0);
	__DELETE(THIS^.pValues);
	END_IF

__DELETE(THIS^.pBuckets);
THIS^._Bucket_Count := 0;
THIS^._Count := 0;
THIS^.bValues_Updated := TRUE;
END_METHOD

// Checks if item is contained in set.
METHOD Contains : BOOL
VAR_INPUT
	Item : ANY; // Item to find.
END_VAR
VAR
	Index : T_Position;
	pCurrent : POINTER TO T_Hashset_Bucket_Node;
END_VAR
Index := THIS^.Hash(Item) MOD THIS^.Bucket_Count;

IF THIS^._Empty THEN RETURN; END_IF

pCurrent := THIS^.pBuckets[Index];

WHILE pCurrent <> 0 DO
	IF F_Compare_Generics(Item, pCurrent^.Data) = T_Comparison.Equal THEN 
		Contains := TRUE;
		THIS^.Clear_Error();
		RETURN; 
		END_IF
	pCurrent := pCurrent^.pNext;
	END_WHILE
END_METHOD

{attribute 'hide'}
METHOD FB_exit : BOOL
VAR_INPUT
	bInCopyCode : BOOL; // if TRUE, the exit method is called for exiting an instance that is copied afterwards (online change).
END_VAR
// Return if it's an online change.
IF bInCopyCode THEN RETURN; END_IF

THIS^.Clear();
END_METHOD

{attribute 'hide'}
METHOD FB_init : BOOL
VAR_INPUT
	bInitRetains : BOOL; // if TRUE, the retain variables are initialized (warm start / cold start)
	bInCopyCode : BOOL;  // if TRUE, the instance afterwards gets moved into the copy code (online change)
	Initial_Bucket_Count : T_Capacity; // Number of buckets you want to initialise the hash set with. Use 0 if you don't know.
END_VAR
// Return if it's an online change.
IF bInCopyCode THEN RETURN; END_IF

THIS^.pBuckets := THIS^.Create_Buckets(Initial_Bucket_Count, Error => THIS^.Error);
THIS^._Bucket_Count := SEL(THIS^.pBuckets <> 0, 0,Initial_Bucket_Count);
END_METHOD

// Gets an immutable list of the values in the set.
METHOD Get_Values : I_Immutable_List
VAR
	i : T_Capacity;
	pCurrent : POINTER TO T_Hashset_Bucket_Node;
END_VAR
IF THIS^.pValues = 0 THEN THIS^.pValues := __NEW(FB_Array_List(Initial_Capacity := 0)); END_IF
THIS^.fbImmutable_Values_List(ipList := THIS^.pValues^);
Get_Values := THIS^.fbImmutable_Values_List;

IF NOT THIS^.bValues_Updated THEN RETURN; END_IF 

pValues^.Clear();

FOR i := 0 TO THIS^._Bucket_Count - 1 DO
	pCurrent := THIS^.pBuckets[i];
	WHILE pCurrent <> 0 DO
		pValues^.Insert_Generic(pValues^._Count, pCurrent^.Data);
		pCurrent := pCurrent^.pNext;
		END_WHILE
	END_FOR
	
THIS^.bValues_Updated := FALSE;
END_METHOD

// Insert item into set.
METHOD Insert : I_Set
VAR_INPUT
	Item : ANY; // Data to insert
END_VAR
VAR_OUTPUT
	bSuccess : BOOL; // Indicates whether operation was successful. Success = TRUE, Failure = FALSE
END_VAR
Insert := THIS^.Insert_Generic(Item, bSuccess => bSuccess);
END_METHOD

// Adds new generic item at into set.
// The set will store a copy of the generic item so as to not modify the original value outside it's scope.
METHOD Insert_Generic : I_Set
VAR_INPUT
	Item : T_Generic; // Item to store
END_VAR
VAR_OUTPUT
	bSuccess 	: BOOL; // Indicates whether operation was successful. Success = TRUE, Failure = FALSE
END_VAR
VAR
	Index : T_Position;
	pCurrent : POINTER TO T_Hashset_Bucket_Node;
END_VAR
Insert_Generic := THIS^;

IF TO_REAL(THIS^._Count) > (TO_REAL(THIS^.Bucket_Count) * THIS^.fLoad_Factor) OR_ELSE THIS^.Bucket_Count <= 0 THEN
	// Increasing the bucket by 50% once the load factor is reached.
	// Bitwise shifting is the same as multiplying by 1.5, this is done because no complicated casting is needed.
	THIS^.Resize(SEL(THIS^.Bucket_Count > 1, 16, THIS^.Bucket_Count + SHR(THIS^.Bucket_Count, 1)), bSuccess => bSuccess);
	IF NOT bSuccess THEN RETURN; END_IF
	END_IF
	
Index := THIS^.Hash(Item) MOD THIS^.Bucket_Count;

pCurrent := THIS^.pBuckets[Index];

WHILE pCurrent <> 0 DO
	IF F_Compare_Generics(Item, pCurrent^.Data) = T_Comparison.Equal THEN RETURN; END_IF
	pCurrent := pCurrent^.pNext;
	END_WHILE
	
pCurrent := THIS^.Create_Node(Item, bSuccess => bSuccess, Error => Error);

IF NOT bSuccess THEN RETURN; END_IF

pCurrent^.pNext := THIS^.pBuckets[Index];
THIS^.pBuckets[Index] := pCurrent;

THIS^.Increment_Count();
THIS^.bValues_Updated := TRUE;
END_METHOD

// Removes item from the set.
METHOD Remove : I_Set
VAR_INPUT
	Item : ANY; // Data to remove
END_VAR
VAR_OUTPUT
	bSuccess : BOOL; // Indicates whether operation was successful. Success = TRUE, Failure = FALSE
END_VAR
Remove := THIS^.Remove_Generic(Item, bSuccess => bSuccess);
END_METHOD

// Removes generic item from the set.
METHOD Remove_Generic : I_Set
VAR_INPUT
	Item : T_Generic; // Data to remove
END_VAR
VAR_OUTPUT
	bSuccess : BOOL; // Indicates whether operation was successful. Success = TRUE, Failure = FALSE
END_VAR
VAR
	Index : T_Position;
	pCurrent, pPrevious : POINTER TO T_Hashset_Bucket_Node;
END_VAR
Remove_Generic := THIS^;

IF THIS^._Empty THEN RETURN; END_IF

Index := THIS^.Hash(Item) MOD THIS^.Bucket_Count;

pCurrent := THIS^.pBuckets[Index];

WHILE pCurrent <> 0 DO
	IF F_Compare_Generics(Item, pCurrent^.Data) = T_Comparison.Equal THEN
		IF pPrevious <> 0 THEN 
			pPrevious^.pNext := pCurrent^.pNext;
		ELSE
			THIS^.pBuckets[Index] := pCurrent^.pNext;
			END_IF
		THIS^.Delete_Node(pCurrent);
		bSuccess := TRUE;
		THIS^.Decrement_Count();
		THIS^.bValues_Updated := TRUE;
		THIS^.Clear_Error();
		RETURN;
		END_IF
		
	pPrevious := pCurrent;
	pCurrent := pCurrent^.pNext;
	END_WHILE
END_METHOD

// Sets the number of buckets in the hash set.
// Existing items are rehashed and redistributed into the new buckets.
// Note that of the count is 0 the hashtable is cleared.
METHOD Resize : I_Hash_Set
VAR_INPUT
	Count : T_Capacity;
END_VAR
VAR_OUTPUT
	bSuccess : BOOL;
END_VAR
VAR
	Hash : DWORD;
	New_Index : T_Position;
	i : T_Capacity;
	pCurrent, pNext : POINTER TO T_Hashset_Bucket_Node;
	pNew_Bucket : POINTER TO POINTER TO T_Hashset_Bucket_Node;
END_VAR
Resize := THIS^;

IF Count < 0 THEN THIS^._Error_Status := GVL_Errors.ERR_INDEX_OUT_OF_BOUNDS; RETURN; END_IF
IF Count = 0 THEN THIS^.Clear(); bSuccess := TRUE; RETURN; END_IF
IF Count = THIS^._Bucket_Count THEN bSuccess := TRUE; RETURN; END_IF

pNew_Bucket := THIS^.Create_Buckets(Count, bSuccess => bSuccess, Error => THIS^.Error);

IF NOT bSuccess THEN RETURN; END_IF

FOR i := 0 TO THIS^._Bucket_Count - 1 DO
	pCurrent := THIS^.pBuckets[i];
	WHILE pCurrent <> 0 DO
		pNext := pCurrent^.pNext;
		New_Index := THIS^.Hash(pCurrent^.Data) MOD Count;
		pCurrent^.pNext := pNew_Bucket[New_Index];
		pNew_Bucket[New_Index] := pCurrent;
		pCurrent := pNext;
		END_WHILE
	END_FOR
	
__DELETE(THIS^.pBuckets);
THIS^.pBuckets := pNew_Bucket;
THIS^._Bucket_Count := Count;
END_METHOD

END_FUNCTION_BLOCK

// POUs/Function Blocks/Collections/FB_Queue
// A collection whose access/mutation of items is first-in, first-out.
{attribute 'enable_dynamic_creation'}
{attribute 'no_assign'}
{attribute 'no_explicit_call' := 'direct call for this function block is not allowed'}
FUNCTION_BLOCK FB_Queue IMPLEMENTS I_Queue//, I_Enumerable, I_Copyable
VAR
	fbList : FB_List := ();
END_VAR

// Number of items in the collection.
PROPERTY _Count : T_Capacity
GET
_Count := THIS^.fbList._Count;
END_GET
END_PROPERTY

// Checks if collection is empty.
PROPERTY _Empty : BOOL
GET
_Empty := THIS^.fbList._Empty;
END_GET
END_PROPERTY

// Error status of the collection.
PROPERTY _Error_Status : T_Error
GET
_Error_Status := THIS^.fbList._Error_Status;
END_GET
END_PROPERTY

// Gets an immutable list of the items in the queue.
PROPERTY _Values : I_Immutable_List
GET
VAR_INST
	fbImmutable_List : FB_Immutable_List := (ipList := THIS^.fbList);
END_VAR
_Values := fbImmutable_List;
END_GET
END_PROPERTY

// Empties/Clears/Deletes every item in the queue.
METHOD Clear : I_Queue
Clear := THIS^;

THIS^.fbList.Clear();
END_METHOD

// Removes item at the front the queue.
METHOD Dequeue : I_Queue
VAR_OUTPUT
	bSuccess : BOOL;
END_VAR
Dequeue := THIS^;

THIS^.fbList.Remove_At(0, bSuccess => bSuccess);
END_METHOD

// Adds item at the back of the queue.
METHOD Enqueue : I_Queue
VAR_INPUT
	Item : ANY; // Variable containg data to store on the queue.
END_VAR
VAR_OUTPUT
	bSuccess : BOOL;
END_VAR
Enqueue := THIS^;

THIS^.fbList.Insert_Generic(THIS^.fbList._Count, Item, bSuccess => bSuccess);
END_METHOD

// Adds item at the front of the queue.
METHOD Enqueue_At_Front : I_Queue
VAR_INPUT
	Item : ANY; // Variable containg data to store on the queue.
END_VAR
VAR_OUTPUT
	bSuccess : BOOL;
END_VAR
Enqueue_At_Front := THIS^;

THIS^.fbList.Insert_Generic(0, Item, bSuccess => bSuccess);
END_METHOD

// Adds a generic item at the back of the queue.
METHOD Enqueue_Generic : I_Queue
VAR_INPUT
	Item : T_Generic; // Item to store.
	bAt_Front : BOOL; // Enqueues at front if set to TRUE.
END_VAR
VAR_OUTPUT
	bSuccess : BOOL;
END_VAR
Enqueue_Generic := THIS^;

IF bAt_Front THEN
	THIS^.fbList.Insert_Generic(0, Item, bSuccess => bSuccess);
ELSE
	THIS^.fbList.Insert_Generic(THIS^.fbList._Count, Item, bSuccess => bSuccess);
	END_IF
END_METHOD

// Gets the item at the front of the queue.
METHOD Get : I_Queue
VAR_INPUT
	Item : ANY; // Variable to store returned item value
END_VAR
VAR_OUTPUT
	bSuccess : BOOL;
END_VAR
Get := THIS^;

THIS^.fbList.Get(0, Item, bSuccess => bSuccess);
END_METHOD

// Gets the item at the front of the queue as a generic.
METHOD Get_Generic : I_Queue
VAR_OUTPUT
	Item : T_Generic; // Variable to store returned item value
	bSuccess : BOOL;
END_VAR
Get_Generic := THIS^;

THIS^.fbList.Get_Generic(0, Item => Item, bSuccess => bSuccess);
END_METHOD

// Reverses the order of the items in the queue.
METHOD Reverse : I_Queue
VAR_OUTPUT
	bSuccess : BOOL;
END_VAR
Reverse := THIS^;

THIS^.fbList.Reverse(bSuccess => bSuccess);
END_METHOD

END_FUNCTION_BLOCK

// POUs/Function Blocks/Collections/FB_Stack
// A collection whose access/mutation of items is last-in, first-out.
{attribute 'enable_dynamic_creation'}
{attribute 'no_assign'}
{attribute 'no_explicit_call' := 'direct call for this function block is not allowed'}
FUNCTION_BLOCK FB_Stack IMPLEMENTS I_Stack //, I_Enumerable, I_Copyable
VAR
	fbList : FB_List;
END_VAR

// Number of items in the collection.
PROPERTY _Count : T_Capacity
GET
_Count := THIS^.fbList._Count;
END_GET
END_PROPERTY

// Checks if collection is empty.
PROPERTY _Empty : BOOL
GET
_Empty := THIS^.fbList._Empty;
END_GET
END_PROPERTY

// Error status of the collection.
PROPERTY _Error_Status : T_Error
GET
_Error_Status := THIS^.fbList._Error_Status;
END_GET
END_PROPERTY

// Gets an immutable list of the items in the stack.
PROPERTY _Values : I_Immutable_List
GET
VAR_INST
	fbImmutable_List : FB_Immutable_List := (ipList := THIS^.fbList);
END_VAR
_Values := fbImmutable_List;
END_GET
END_PROPERTY

// Empties/Clears/Deletes every item in the stack.
METHOD Clear : I_Stack
Clear := THIS^;

THIS^.fbList.Clear();
END_METHOD

// Gets item at the top of the stack.
METHOD Get : I_Stack
VAR_INPUT
	Item : ANY; // Variable to store returned item value. 
END_VAR
VAR_OUTPUT
	bSuccess : BOOL;
END_VAR
Get := THIS^;

THIS^.fbList.Get(0, Item, bSuccess => bSuccess);
END_METHOD

// Gets item at the top of the stack as a generic.
METHOD Get_Generic : I_Stack
VAR_OUTPUT
	Item : T_Generic; // Variable to store returned item value
	bSuccess : BOOL;
END_VAR
Get_Generic := THIS^;

THIS^.fbList.Get_Generic(0, Item => Item, bSuccess => bSuccess);
END_METHOD

// Removes item at the top of the stack without returning anything.
METHOD Pop : I_Stack
VAR_OUTPUT
	bSuccess : BOOL;
END_VAR
Pop := THIS^;

THIS^.fbList.Remove_At(0, bSuccess => bSuccess);
END_METHOD

// Add item to the top of the stack.
METHOD Push : I_Stack
VAR_INPUT
	Item : ANY; // Item to store.
END_VAR
VAR_OUTPUT
	bSuccess : BOOL;
END_VAR
Push := THIS^;

THIS^.fbList.Insert_Generic(0, Item, bSuccess => bSuccess);
END_METHOD

// Add generic item to the top of the stack.
METHOD Push_Generic : I_Stack
VAR_INPUT
	Item : T_Generic; // Item to store.
END_VAR
VAR_OUTPUT
	bSuccess : BOOL;
END_VAR
Push_Generic := THIS^;

THIS^.fbList.Insert_Generic(0, Item, bSuccess => bSuccess);
END_METHOD

// Reverses order of items on stack.
METHOD Reverse : I_Stack
VAR_OUTPUT
	bSuccess : BOOL;
END_VAR
Reverse := THIS^;

THIS^.fbList.Reverse(bSuccess => bSuccess);
END_METHOD

END_FUNCTION_BLOCK

// POUs/Function Blocks/Collections/FB_Tree_Map
// A collection of key-value pair items implemented using an iterative AVL Tree. 
// Keys and values can be retrieved as an immutable list (whose base is FB_ArrayList) via 4 traversal methods; Inorder, Preorder, Postorder and Level Order.
// This data structure was implemented with the help of Max Goren's iterative AVL tree in C++. See Function Block's body for more details.
{attribute 'enable_dynamic_creation'}
{attribute 'no_assign'}
{attribute 'no_explicit_call' := 'direct call for this function block is not allowed'}
FUNCTION_BLOCK FB_Tree_Map EXTENDS FB_Collection IMPLEMENTS I_Tree_Map //, I_Enumerable, I_Copyable
VAR
	pRoot : POINTER TO T_AVL_Map_Node;
	Traversal : T_BST_Traversal := T_BST_Traversal.In_Order; 
	pKeys, pValues : POINTER TO FB_Array_List;
	fbImmutable_Keys_List,
	fbImmutable_Values_List : FB_Immutable_List;
	bKeys_Updated, bValues_Updated : BOOL := TRUE;
END_VAR

(*
	https://github.com/maxgoren
	https://github.com/maxgoren/Algorithms/
	http://www.maxgcoding.com/iterative-avl-trees-insertion/
	http://www.maxgcoding.com/iterative-avl-trees-deletion/

	MIT License
	
	Copyright (c) 2021 Max Goren
	
	Permission is hereby granted, free of charge, to any person obtaining a copy
	of this software and associated documentation files (the "Software"), to deal
	in the Software without restriction, including without limitation the rights
	to use, copy, modify, merge, publish, distribute, sublicense, and/or sell
	copies of the Software, and to permit persons to whom the Software is
	furnished to do so, subject to the following conditions:
	
	The above copyright notice and this permission notice shall be included in all
	copies or substantial portions of the Software.
	
	THE SOFTWARE IS PROVIDED "AS IS", WITHOUT WARRANTY OF ANY KIND, EXPRESS OR
	IMPLIED, INCLUDING BUT NOT LIMITED TO THE WARRANTIES OF MERCHANTABILITY,
	FITNESS FOR A PARTICULAR PURPOSE AND NONINFRINGEMENT. IN NO EVENT SHALL THE
	AUTHORS OR COPYRIGHT HOLDERS BE LIABLE FOR ANY CLAIM, DAMAGES OR OTHER
	LIABILITY, WHETHER IN AN ACTION OF CONTRACT, TORT OR OTHERWISE, ARISING FROM,
	OUT OF OR IN CONNECTION WITH THE SOFTWARE OR THE USE OR OTHER DEALINGS IN THE
	SOFTWARE.
*)

// Performs rotation and updates heights until tree is balanced.
METHOD PROTECTED Balance
VAR_INPUT
    pNode : POINTER TO T_AVL_Map_Node;
END_VAR
VAR 
    Balance_Factor : T_Position;
END_VAR
WHILE pNode <> 0 DO
	THIS^.Update_Height(pNode);
	
	Balance_Factor := THIS^.Get_Balance(pNode);
	
	IF Balance_Factor < -1 THEN
		IF THIS^.Get_Balance(pNode^.pRight) > 0 THEN THIS^.Rotate_Right(pNode^.pRight); END_IF
		THIS^.Rotate_Left(pNode);
	ELSIF Balance_Factor > 1 THEN
		IF THIS^.Get_Balance(pNode^.pLeft) < 0 THEN THIS^.Rotate_Left(pNode^.pLeft); END_IF
		THIS^.Rotate_Right(pNode);
		END_IF
		
	pNode := pNode^.pParent;
	END_WHILE
END_METHOD

// Deletes the node and its tree/sub-trees.
{warning disable C0394}
METHOD PROTECTED Clear_Node
VAR_INPUT
	pRoot : POINTER TO T_AVL_Map_Node;
END_VAR
VAR
	fbNode_Stack : FB_Stack;
	pTmp : POINTER TO T_AVL_Map_Node;
END_VAR
IF pRoot = 0 THEN RETURN; END_IF

fbNode_Stack.Push(pRoot);

WHILE NOT fbNode_Stack._Empty DO
	fbNode_Stack.Get(pTmp).Pop();
	
	IF pTmp^.pRight <> 0 THEN fbNode_Stack.Push(pTmp^.pRight); END_IF
	IF pTmp^.pLeft <> 0 THEN fbNode_Stack.Push(pTmp^.pLeft); END_IF
	
	THIS^.Delete_Node(pTmp);
	END_WHILE
END_METHOD

// Creates a new node in dynamic memory with a clone of the generic item as it data.
METHOD PROTECTED Create_Node : POINTER TO ST_AVL_MAP_NODE
VAR_INPUT
	Key, Value : T_Generic;
END_VAR
VAR_OUTPUT
	bSuccess : BOOL;
	Error : T_Error;
END_VAR
Create_Node := __NEW(ST_AVL_MAP_NODE);

IF Create_Node = 0 THEN Error := GVL_Errors.ERR_MALLOC_FAILED; RETURN; END_IF

Create_Node^.Key := F_Clone_Generic(Key, bSuccess => bSuccess, Error => Error);

IF NOT bSuccess THEN 
	__DELETE(Create_Node);
	RETURN;
	END_IF

Create_Node^.Value := F_Clone_Generic(Value, bSuccess => bSuccess, Error => Error);

IF NOT bSuccess THEN 
	F_Delete_Generic(Create_Node^.Key);
	__DELETE(Create_Node);
	END_IF
END_METHOD

// Safety deletes node.
// If the node and/or it's value/data is in dynamic memory it/they will be deleted.
METHOD PROTECTED Delete_Node
VAR_INPUT
	pNode : REFERENCE TO POINTER TO T_AVL_Map_Node;
END_VAR
IF (pNode = 0) THEN RETURN; END_IF 

F_Delete_Generic(pNode^.Key);
F_Delete_Generic(pNode^.Value);

CASE Tc2_System.F_CheckMemoryArea(pNode, 1) OF
	Tc2_System.E_TcMemoryArea.Dynamic: __DELETE(pNode);
ELSE
	pNode := 0;
	END_CASE
END_METHOD

// Finds the node with the smallest item in a tree or sub-tree.
METHOD PROTECTED Find_Minimum_Node : POINTER TO T_AVL_Node
VAR_INPUT
	pNode : POINTER TO T_AVL_Map_Node;
END_VAR
IF pNode = 0 THEN RETURN; END_IF

WHILE pNode^.pLeft <> 0 DO
	pNode := pNode^.pLeft;
	END_WHILE
	
Find_Minimum_Node := pNode;
END_METHOD

// Gets the difference between the left and right sub-trees.
METHOD PROTECTED Get_Balance : T_Position
VAR_INPUT
	pNode : POINTER TO T_AVL_Map_Node;
END_VAR
Get_Balance :=  THIS^.Get_Height(pNode^.pLeft) - THIS^.Get_Height(pNode^.pRight);
END_METHOD

// Safely gets the height of a sub-tree.
METHOD PROTECTED Get_Height : T_Position
VAR_INPUT
	pNode : POINTER TO T_AVL_Map_Node;
END_VAR
Get_Height := SEL(pNode <> 0, -1, pNode^.Height);
END_METHOD

// Moves from node at source into the position of the destination.
METHOD PROTECTED Move_Node
VAR_INPUT
	pDestination, pSource : POINTER TO T_AVL_Map_Node;
END_VAR
IF pDestination = 0 OR_ELSE pSource = 0 THEN RETURN; END_IF 

IF pDestination^.pParent = 0 THEN
	THIS^.pRoot := pSource;
ELSIF pDestination = pDestination^.pParent^.pLeft THEN
	pDestination^.pParent^.pLeft := pSource;
ELSE
	pDestination^.pParent^.pRight := pSource;
	END_IF
	
IF pSource <> 0 THEN
	pSource^.pParent := pDestination^.pParent;
	END_IF
END_METHOD

// Finds and removes a node from a tree/sub-tree and returns the new root of the tree/subtree.
METHOD PROTECTED Remove_Node : POINTER TO T_AVL_Map_Node
VAR_INPUT
	pNode : REFERENCE TO POINTER TO T_AVL_Map_Node;
END_VAR
VAR
	pSuccessor : POINTER TO T_AVL_Map_Node;
END_VAR
IF (NOT __ISVALIDREF(pNode)) OR_ELSE pNode = 0 THEN RETURN; END_IF 

IF pNode^.pLeft = 0 THEN
	THIS^.Move_Node(pNode, pNode^.pRight);
	Remove_Node := pNode^.pRight;
ELSIF pNode^.pRight = 0 THEN 
	THIS^.Move_Node(pNode, pNode^.pLeft);
	Remove_Node := pNode^.pLeft;
ELSE
	Remove_Node := pSuccessor := THIS^.Find_Minimum_Node(pNode^.pRight);
	IF pSuccessor^.pParent <> pNode THEN 
		THIS^.Move_Node(pSuccessor, pSuccessor^.pRight);
		pSuccessor^.pRight := pNode^.pRight;
		pSuccessor^.pRight^.pParent := pSuccessor;
		END_IF
	THIS^.Move_Node(pNode, pSuccessor);
	pSuccessor^.pLeft := pNode^.pLeft;
	pSuccessor^.pLeft^.pParent := pSuccessor;
	END_IF

THIS^.Delete_Node(pNode);
END_METHOD

// Rotates a tree/sub-tree left.
METHOD PROTECTED Rotate_Left
VAR_INPUT
    pX : POINTER TO T_AVL_Map_Node;
END_VAR
VAR
    pY : POINTER TO T_AVL_Map_Node := pX^.pRight;
END_VAR
IF pY <> 0 THEN
	pX^.pRight := pY^.pLeft;
	IF pY^.pLeft <> 0 THEN pY^.pLeft^.pParent := pX; END_IF
	pY^.pParent := pX^.pParent;
	END_IF
	
IF pX^.pParent = 0 THEN
	THIS^.pRoot := pY;
ELSIF pX = pX^.pParent^.pLeft THEN
	pX^.pParent^.pLeft := pY;
ELSE
	pX^.pParent^.pRight := pY;
	END_IF
	
IF pY <> 0 THEN pY^.pLeft := pX; END_IF
	
pX^.pParent := pY;
THIS^.Update_Height(pX);
THIS^.Update_Height(pY);
END_METHOD

// Rotates a tree/sub-tree right.
METHOD PROTECTED Rotate_Right
VAR_INPUT
    pX : POINTER TO T_AVL_Map_Node;
END_VAR
VAR
    pY : POINTER TO T_AVL_Map_Node := pX^.pLeft;
END_VAR
IF pY <> 0 THEN
	pX^.pLeft := pY^.pRight;
	IF pY^.pRight <> 0 THEN pY^.pRight^.pParent := pX; END_IF
	pY^.pParent := pX^.pParent;
	END_IF
	
IF pX^.pParent = 0 THEN
	THIS^.pRoot := pY;
ELSIF pX = pX^.pParent^.pLeft THEN
	pX^.pParent^.pLeft := pY;
ELSE
	pX^.pParent^.pRight := pY;
	END_IF
	
IF pY <> 0 THEN pY^.pRight := pX; END_IF
	
pX^.pParent := pY;
THIS^.Update_Height(pX);
THIS^.Update_Height(pY);
END_METHOD

// Checks if an item is in a tree/ sub-tree.
METHOD PROTECTED Search_Node : POINTER TO T_AVL_Map_Node
VAR_INPUT
	pNode : POINTER TO T_AVL_Map_Node;
	Key : T_Generic;
END_VAR
WHILE pNode <> 0 DO
	CASE F_Compare_Generics(Key, pNode^.Key) OF
		T_Comparison.Less	: pNode := pNode^.pLeft;
		T_Comparison.Greater: pNode := pNode^.pRight; 
		T_Comparison.Equal	: 
			Search_Node := pNode;
			RETURN;
		END_CASE
	END_WHILE
END_METHOD

METHOD PROTECTED Update_Height
VAR_INPUT
	pNode : POINTER TO T_AVL_Map_Node;
END_VAR
IF pNode = 0 THEN RETURN; END_IF
pNode^.Height := 1 + MAX(THIS^.Get_Height(pNode^.pLeft), THIS^.Get_Height(pNode^.pRight));
END_METHOD

// Traversal method for retrieving keys and values in the tree map set.
PROPERTY _Traversal : T_BST_Traversal
GET
_Traversal := THIS^.Traversal;
END_GET
SET
IF THIS^.Traversal <> _Traversal THEN 
	THIS^.bKeys_Updated := THIS^.bValues_Updated := TRUE;
	END_IF

THIS^.Traversal := _Traversal;
END_SET
END_PROPERTY

// Empties/Clears/Deletes every item in the map.
METHOD Clear : I_Map
Clear := THIS^;

THIS^.Clear_Node(THIS^.pRoot);

IF THIS^.pKeys <> 0 THEN 
	THIS^.fbImmutable_Keys_List(ipList := 0); 
	__DELETE(THIS^.pKeys); END_IF

IF THIS^.pValues <> 0 THEN
	THIS^.fbImmutable_Values_List(ipList := 0);
	__DELETE(THIS^.pValues);
	END_IF

THIS^.pRoot := 0;
THIS^._Count := 0;
THIS^.bKeys_Updated := THIS^.bValues_Updated := TRUE;
END_METHOD

// Checks if key is contained in the map.
METHOD Contains : BOOL
VAR_INPUT
	Key : ANY; // Key to find.
END_VAR
Contains := THIS^.Search_Node(THIS^.pRoot, Key) <> 0;
END_METHOD

{attribute 'hide'}
METHOD FB_exit : BOOL
VAR_INPUT
	bInCopyCode : BOOL; // if TRUE, the exit method is called for exiting an instance that is copied afterwards (online change).
END_VAR
// If this is an online change or this collection is empty then ignore. 
IF bInCopyCode THEN RETURN; END_IF

THIS^.Clear();
END_METHOD

// Gets the value associated with the specified key without removing it from the map.
METHOD Get : I_Map
VAR_INPUT
	Key : ANY; // Key used to identify stored value
	Value : ANY; // Variable to store requested data 
END_VAR
VAR_OUTPUT
	bSuccess : BOOL;
END_VAR
VAR
	Tmp : T_Generic;
END_VAR
Get := THIS^;

THIS^.Get_Generic(Key, Value => Tmp, bSuccess => bSuccess);

IF NOT bSuccess THEN RETURN; END_IF

IF NOT F_Matching_Generics(Value, Tmp) THEN
	THIS^._Error_Status := GVL_Errors.ERR_TYPE_MISMATCH;
	RETURN;
	END_IF
	
F_Copy_Generic_Value(Tmp, Value, bSuccess => bSuccess, Error => Error);
END_METHOD

// Returns value as a string, if type to string conversion is supported.
METHOD Get_As_String : I_Map
VAR_INPUT
	Key : ANY; // Key used to identify stored value
	sValue : REFERENCE TO STRING; // Variable to store returned item.
END_VAR
VAR_OUTPUT
	bSuccess : BOOL;
END_VAR
VAR
	Tmp : T_Generic;
END_VAR
Get_As_String := THIS^;

IF NOT __ISVALIDREF(sValue) THEN 
	THIS^._Error_Status := GVL_Errors.ERR_INVALID_REFERENCE;
	RETURN;
	END_IF
	
THIS^.Get_Generic(Key, Value => Tmp, bSuccess => bSuccess);

IF NOT bSuccess THEN RETURN; END_IF
	
CASE Tmp.TypeClass OF
	T_Type.TYPE_STRING:
		Tc2_Utilities.STRNCPY(ADR(sValue), Tmp.pValue, MIN(Tc2_Utilities.LEN2(ADR(sValue))+1, TO_UDINT(Tmp.diSize)));
		THIS^.Clear_Error();

	T_Type.TYPE_WSTRING:
		Tc2_Utilities.WSTRING_TO_STRING2(ADR(sValue), Tmp.pValue, MIN(Tc2_Utilities.LEN2(ADR(sValue))+1, TO_UDINT(Tmp.diSize)));
		THIS^.Clear_Error();
ELSE
	sValue := F_Generic_To_String(Tmp, bSuccess => bSuccess, Error => THIS^.Error);
	END_CASE
END_METHOD

// Gets the value in its generic form associated with the specified key in its generic form without removing it from the map.
// (** Use carefully as this contains the pointer of the actual value in the collection. **)
// If you wish to use this it is recommeded you create a copy of the returned value using MEMMOVE or MEMCPY
METHOD Get_Generic : I_Map
VAR_INPUT
	Key : T_Generic; // Key used to identify stored value
END_VAR
VAR_OUTPUT
	Value : T_Generic := (TypeClass := T_Type.TYPE_NONE); // Variable to store requested data 
	bSuccess : BOOL;
END_VAR
VAR
	pTmp : POINTER TO T_AVL_Map_Node;
END_VAR
Get_Generic := THIS^;

pTmp := THIS^.Search_Node(THIS^.pRoot, Key);
bSuccess := pTmp <> 0;

IF NOT bSuccess THEN 
	// Throw item not found error.
	THIS^._Error_Status := GVL_Errors.ERR_NO_KEY;
	RETURN; 
	END_IF

Value := pTmp^.Value;
END_METHOD

// Gets an immutable list of the keys.
{warning disable C0394}
METHOD Get_Keys : I_Immutable_List
VAR
	pCurrent : POINTER TO T_AVL_Map_Node := THIS^.pRoot;
	pPrevious, pTmp : POINTER TO T_AVL_Map_Node;
	fbNode_Buffer : FB_Queue;
	bSuccess : BOOL;
END_VAR
IF THIS^.pKeys = 0 THEN THIS^.pKeys := __NEW(FB_Array_List(Initial_Capacity := 0)); END_IF
THIS^.fbImmutable_Keys_List(ipList := THIS^.pKeys^);
Get_Keys := THIS^.fbImmutable_Keys_List;

IF NOT THIS^.bKeys_Updated THEN RETURN; END_IF

THIS^.pKeys^.Clear();

IF pCurrent = 0 THEN RETURN; END_IF

WHILE (NOT fbNode_Buffer._Empty) OR_ELSE pCurrent <> 0 DO
	
	CASE THIS^._Traversal OF
		T_BST_Traversal.In_Order:
			IF pCurrent <> 0 THEN 
				fbNode_Buffer.Enqueue_At_Front(pCurrent);
				pCurrent := pCurrent^.pLeft;
			ELSE
				fbNode_Buffer.Get(pCurrent).Dequeue();
				THIS^.pKeys^.Insert_Generic(THIS^.pKeys^._Count, pCurrent^.Key);
				pCurrent := pCurrent^.pRight;
				END_IF
				
		T_BST_Traversal.Pre_Order:
			IF pCurrent <> 0 THEN 
				THIS^.pKeys^.Insert_Generic(THIS^.pKeys^._Count, pCurrent^.Key);
				IF pCurrent^.pRight <> 0 THEN fbNode_Buffer.Enqueue_At_Front(pCurrent^.pRight); END_IF
				pCurrent := pCurrent^.pLeft;
			ELSE
				fbNode_Buffer.Get(pCurrent).Dequeue();
				END_IF
			
		T_BST_Traversal.Post_Order:
			WHILE pCurrent <> 0 DO 
				fbNode_Buffer.Enqueue_At_Front(pCurrent);
				pCurrent := pCurrent^.pLeft;
				END_WHILE
				
			IF NOT fbNode_Buffer._Empty THEN
				fbNode_Buffer.Get(pTmp);
				pTmp := pTmp^.pRight;
				IF pTmp = 0 OR_ELSE pTmp = pPrevious THEN 
					fbNode_Buffer.Get(pCurrent).Dequeue();
					THIS^.pKeys^.Insert_Generic(THIS^.pKeys^._Count, pCurrent^.Key);
					pPrevious := pCurrent;
					pCurrent := 0;
				ELSE
					pCurrent := pTmp;
					END_IF
				END_IF
			
		T_BST_Traversal.Level_Order:
			THIS^.pKeys^.Insert_Generic(THIS^.pKeys^._Count, pCurrent^.Key);
			IF pCurrent^.pLeft <> 0 THEN fbNode_Buffer.Enqueue(pCurrent^.pLeft); END_IF
			IF pCurrent^.pRight <> 0 THEN fbNode_Buffer.Enqueue(pCurrent^.pRight); END_IF
			fbNode_Buffer.Get(pCurrent).Dequeue(bSuccess => bSuccess);
			IF NOT bSuccess THEN pCurrent := 0; END_IF
	ELSE
		EXIT;
		END_CASE
	END_WHILE
	
THIS^.bKeys_Updated := FALSE;
END_METHOD

// Gets an immutable list of the values.
{warning disable C0394}
METHOD Get_Values : I_Immutable_List
VAR
	pCurrent : POINTER TO T_AVL_Map_Node := THIS^.pRoot;
	pPrevious, pTmp : POINTER TO T_AVL_Map_Node;
	fbNode_Buffer : FB_Queue;
	bSuccess : BOOL;
END_VAR
IF THIS^.pValues = 0 THEN THIS^.pValues := __NEW(FB_Array_List(Initial_Capacity := 0)); END_IF
THIS^.fbImmutable_Values_List(ipList := THIS^.pValues^);
Get_Values := THIS^.fbImmutable_Values_List;

IF NOT THIS^.bValues_Updated THEN RETURN; END_IF

THIS^.pValues^.Clear();

IF pCurrent = 0 THEN RETURN; END_IF

WHILE (NOT fbNode_Buffer._Empty) OR_ELSE pCurrent <> 0 DO
	
	CASE THIS^._Traversal OF
		T_BST_Traversal.In_Order:
			IF pCurrent <> 0 THEN 
				fbNode_Buffer.Enqueue_At_Front(pCurrent);
				pCurrent := pCurrent^.pLeft;
			ELSE
				fbNode_Buffer.Get(pCurrent).Dequeue();
				THIS^.pValues^.Insert_Generic(THIS^.pValues^._Count, pCurrent^.Value);
				pCurrent := pCurrent^.pRight;
				END_IF
				
		T_BST_Traversal.Pre_Order:
			IF pCurrent <> 0 THEN 
				THIS^.pValues^.Insert_Generic(THIS^.pValues^._Count, pCurrent^.Value);
				IF pCurrent^.pRight <> 0 THEN fbNode_Buffer.Enqueue_At_Front(pCurrent^.pRight); END_IF
				pCurrent := pCurrent^.pLeft;
			ELSE
				fbNode_Buffer.Get(pCurrent).Dequeue();
				END_IF
			
		T_BST_Traversal.Post_Order:
			WHILE pCurrent <> 0 DO 
				fbNode_Buffer.Enqueue_At_Front(pCurrent);
				pCurrent := pCurrent^.pLeft;
				END_WHILE
				
			IF NOT fbNode_Buffer._Empty THEN
				fbNode_Buffer.Get(pTmp);
				pTmp := pTmp^.pRight;
				IF pTmp = 0 OR_ELSE pTmp = pPrevious THEN 
					fbNode_Buffer.Get(pCurrent).Dequeue();
					THIS^.pValues^.Insert_Generic(THIS^.pValues^._Count, pCurrent^.Value);
					pPrevious := pCurrent;
					pCurrent := 0;
				ELSE
					pCurrent := pTmp;
					END_IF
				END_IF
			
		T_BST_Traversal.Level_Order:
			THIS^.pValues^.Insert_Generic(THIS^.pValues^._Count, pCurrent^.Value);
			IF pCurrent^.pLeft <> 0 THEN fbNode_Buffer.Enqueue(pCurrent^.pLeft); END_IF
			IF pCurrent^.pRight <> 0 THEN fbNode_Buffer.Enqueue(pCurrent^.pRight); END_IF
			fbNode_Buffer.Get(pCurrent).Dequeue(bSuccess => bSuccess);
			IF NOT bSuccess THEN pCurrent := 0; END_IF
	ELSE
		EXIT;
		END_CASE
	END_WHILE
	
THIS^.bValues_Updated := FALSE;
END_METHOD

// Insert an element with the provided key and value to the map.
METHOD Insert : I_Map
VAR_INPUT
	Key : ANY; // Key used to identify stored value
	Value : ANY; // Value to store in map with key
END_VAR
VAR_OUTPUT
	bSuccess : BOOL;
END_VAR
Insert := THIS^.Insert_Generic(Key, Value, FALSE, bSuccess => bSuccess);
END_METHOD

// Insert an element with the provided key and value in their generic forms to the map.
METHOD Insert_Generic : I_Map
VAR_INPUT
	Key : T_Generic; // Key used to identify stored value
	Value : T_Generic; // Value to store in map with key
	bUpdate : BOOL; // If this is true the value will be updated if the key already exists.
END_VAR
VAR_OUTPUT
	bSuccess : BOOL;
END_VAR
VAR
	pCurrent, pPrevious : POINTER TO T_AVL_Map_Node;
	Tmp : T_Generic;
END_VAR
Insert_Generic := THIS^;

pCurrent := THIS^.pRoot;
pPrevious := pCurrent;

WHILE pCurrent <> 0 DO
	pPrevious := pCurrent;
	CASE F_Compare_Generics(Key, pCurrent^.Key) OF
		T_Comparison.Less 	 : pCurrent := pCurrent^.pLeft;
		T_Comparison.Greater : pCurrent := pCurrent^.pRight;
		T_Comparison.Equal 	 : 
			IF bUpdate THEN
				Tmp := F_Clone_Generic(Value, bSuccess => bSuccess, Error => THIS^.Error);
				IF NOT bSuccess THEN RETURN; END_IF
				F_Delete_Generic(pCurrent^.Value);
				pCurrent^.Value := Tmp;
				THIS^.bValues_Updated := TRUE;
			ELSE
				THIS^._Error_Status := GVL_Errors.ERR_DUPLICATE_KEY;
				END_IF
			RETURN;
	ELSE
		THIS^._Error_Status := GVL_Errors.ERR_INVALID_COMPARISON;
		RETURN;
		END_CASE
	END_WHILE
	
pCurrent := THIS^.Create_Node(Key, Value, bSuccess => bSuccess, Error => THIS^.Error);

IF NOT bSuccess THEN RETURN; END_IF

IF pPrevious = 0 THEN
	THIS^.pRoot := pCurrent;
ELSE
	CASE F_Compare_Generics(Key, pPrevious^.Key) OF
		T_Comparison.Less: pPrevious^.pLeft := pCurrent;
	ELSE
		pPrevious^.pRight := pCurrent;
		END_CASE
	END_IF
	
pCurrent^.pParent := pPrevious;
	
THIS^.Balance(pCurrent);
THIS^.Increment_Count();
THIS^.bKeys_Updated := THIS^.bValues_Updated := TRUE;
END_METHOD

// Removes value with the specified key from the map.
METHOD Remove : I_Map
VAR_INPUT
	Key : ANY; // Key used to identify stored value
END_VAR
VAR_OUTPUT
	bSuccess : BOOL;
END_VAR
Remove := THIS^.Remove_Generic(Key, bSuccess => bSuccess);
END_METHOD

// Removes value with the specified key in its generic form from the map.
METHOD Remove_Generic : I_Map
VAR_INPUT
	Key : T_Generic; // Key used to identify stored value
END_VAR
VAR_OUTPUT
	bSuccess : BOOL; // Indicates whether operation was successful. Success = TRUE, Failure = FALSE
END_VAR
VAR
	pTmp : POINTER TO T_AVL_Map_Node;
END_VAR
Remove_Generic := THIS^;

pTmp := THIS^.Search_Node(THIS^.pRoot, Key);

IF pTmp = 0 THEN
	THIS^._Error_Status := GVL_Errors.ERR_NO_KEY;
	RETURN;
	END_IF

THIS^.Balance(THIS^.Remove_Node(pTmp));

THIS^.Decrement_Count();
THIS^.Clear_Error();

IF THIS^._Empty THEN THIS^.pRoot := 0; END_IF

bSuccess := TRUE;
THIS^.bKeys_Updated := THIS^.bValues_Updated := TRUE;
END_METHOD

// Updates the value at the provided key with the new value in the map.
METHOD Update : I_Map
VAR_INPUT
	Key 	: ANY; // Key used to identify stored value
	Value 	: ANY; // Value to store in map with key
END_VAR
VAR_OUTPUT
	bSuccess : BOOL;
END_VAR
VAR
	pTmp : POINTER TO T_AVL_Map_Node;
END_VAR
Update := THIS^.Update_Generic(Key, Value, bSuccess => bSuccess);
END_METHOD

// Updates the value at the provided key with the new value in their generic forms in the map.
METHOD Update_Generic : I_Map
VAR_INPUT
	Key 	: T_Generic; // Key used to identify stored value
	Value 	: T_Generic; // Value to store in map with key
END_VAR
VAR_OUTPUT
	bSuccess : BOOL;
END_VAR
VAR
	pTmp : POINTER TO T_AVL_Map_Node;
	Tmp : T_Generic;
END_VAR
Update_Generic := THIS^;

pTmp := THIS^.Search_Node(THIS^.pRoot, Key);

bSuccess := pTmp <> 0;

IF NOT bSuccess THEN 
	THIS^._Error_Status := GVL_Errors.ERR_NO_KEY;
	RETURN;
	END_IF
	
Tmp := F_Clone_Generic(Value, bSuccess => bSuccess, Error => THIS^.Error);

IF NOT bSuccess THEN RETURN; END_IF

F_Delete_Generic(pTmp^.Value);
pTmp^.Value := Tmp;
THIS^.bValues_Updated := TRUE;
END_METHOD

// Updates a value in the map for a given key. If the key doesnt exist, it will be inserted.
METHOD Upsert : I_Map
VAR_INPUT
	Key 	: ANY; // Key used to identify stored value
	Value 	: ANY; // Value to store in map with key
END_VAR
VAR_OUTPUT
	bSuccess : BOOL;
END_VAR
Upsert := THIS^.Insert_Generic(Key, Value, TRUE, bSuccess => bSuccess);
END_METHOD

END_FUNCTION_BLOCK

// POUs/Function Blocks/Collections/FB_Tree_Multiset
// A collection similiar to a set except it allows for duplicate items. It is implemented using an iterative AVL Tree.
// This data structure was implemented with the help of Max Goren's iterative AVL tree in C++. See Function Block's body for more details.
{attribute 'enable_dynamic_creation'}
{attribute 'no_assign'}
{attribute 'no_explicit_call' := 'direct call for this function block is not allowed'}
FUNCTION_BLOCK FB_Tree_Multiset EXTENDS FB_Tree_Set
VAR
END_VAR

(*
	https://github.com/maxgoren
	http://www.maxgcoding.com/iterative-avl-trees-insertion/
	http://www.maxgcoding.com/iterative-avl-trees-deletion/

	MIT License
	
	Copyright (c) 2023 Max Goren
	
	Permission is hereby granted, free of charge, to any person obtaining a copy
	of this software and associated documentation files (the "Software"), to deal
	in the Software without restriction, including without limitation the rights
	to use, copy, modify, merge, publish, distribute, sublicense, and/or sell
	copies of the Software, and to permit persons to whom the Software is
	furnished to do so, subject to the following conditions:
	
	The above copyright notice and this permission notice shall be included in all
	copies or substantial portions of the Software.
	
	THE SOFTWARE IS PROVIDED "AS IS", WITHOUT WARRANTY OF ANY KIND, EXPRESS OR
	IMPLIED, INCLUDING BUT NOT LIMITED TO THE WARRANTIES OF MERCHANTABILITY,
	FITNESS FOR A PARTICULAR PURPOSE AND NONINFRINGEMENT. IN NO EVENT SHALL THE
	AUTHORS OR COPYRIGHT HOLDERS BE LIABLE FOR ANY CLAIM, DAMAGES OR OTHER
	LIABILITY, WHETHER IN AN ACTION OF CONTRACT, TORT OR OTHERWISE, ARISING FROM,
	OUT OF OR IN CONNECTION WITH THE SOFTWARE OR THE USE OR OTHER DEALINGS IN THE
	SOFTWARE.
*)

// Adds new generic item at into set.
// The set will store a copy of the generic item so as to not modify the original value outside it's scope.
METHOD Insert_Generic : I_Set
VAR_INPUT
	Item : T_Generic; // Item to store
END_VAR
VAR_OUTPUT
	bSuccess : BOOL; // Indicates whether operation was successful. Success = TRUE, Failure = FALSE
END_VAR
VAR
	pCurrent, pPrevious : POINTER TO T_AVL_Node;
END_VAR
Insert_Generic := THIS^;

pCurrent := THIS^.pRoot;
pPrevious := pCurrent;

WHILE pCurrent <> 0 DO
	pPrevious := pCurrent;
	CASE F_Compare_Generics(Item, pCurrent^.Data) OF
		T_Comparison.Less 	 : pCurrent := pCurrent^.pLeft;
		T_Comparison.Greater,
		T_Comparison.Equal 	 : pCurrent := pCurrent^.pRight;
	ELSE
		THIS^._Error_Status := GVL_Errors.ERR_INVALID_COMPARISON;
		RETURN;
		END_CASE
	END_WHILE

pCurrent := THIS^.Create_Node(Item, bSuccess => bSuccess, Error => THIS^.Error);

IF NOT bSuccess THEN RETURN; END_IF

IF pPrevious = 0 THEN
	THIS^.pRoot := pCurrent;
ELSE
	CASE F_Compare_Generics(Item, pPrevious^.Data) OF
		T_Comparison.Less: pPrevious^.pLeft := pCurrent;
	ELSE
		pPrevious^.pRight := pCurrent;
		END_CASE
	END_IF

pCurrent^.pParent := pPrevious;
	
THIS^.Balance(pCurrent);
THIS^.Increment_Count();
END_METHOD

END_FUNCTION_BLOCK

// POUs/Function Blocks/Collections/FB_Tree_Set
// A collection that contains no duplicate items implemented using an iterative AVL Tree.
// This data structure was implemented with the help of Max Goren's iterative AVL tree in C++. See Function Block's body for more details.
{attribute 'enable_dynamic_creation'}
{attribute 'no_assign'}
{attribute 'no_explicit_call' := 'direct call for this function block is not allowed'}
FUNCTION_BLOCK FB_Tree_Set EXTENDS FB_Collection IMPLEMENTS I_Tree_Set //, I_Enumerable, I_Copyable
VAR
	pRoot : POINTER TO T_AVL_Node;
	Traversal : T_BST_Traversal := T_BST_Traversal.In_Order; 
	pValues : POINTER TO FB_Array_List;
	fbImmutable_Values_List : FB_Immutable_List;
END_VAR

(*
	https://github.com/maxgoren
	http://www.maxgcoding.com/iterative-avl-trees-insertion/
	http://www.maxgcoding.com/iterative-avl-trees-deletion/

	MIT License
	
	Copyright (c) 2023 Max Goren
	
	Permission is hereby granted, free of charge, to any person obtaining a copy
	of this software and associated documentation files (the "Software"), to deal
	in the Software without restriction, including without limitation the rights
	to use, copy, modify, merge, publish, distribute, sublicense, and/or sell
	copies of the Software, and to permit persons to whom the Software is
	furnished to do so, subject to the following conditions:
	
	The above copyright notice and this permission notice shall be included in all
	copies or substantial portions of the Software.
	
	THE SOFTWARE IS PROVIDED "AS IS", WITHOUT WARRANTY OF ANY KIND, EXPRESS OR
	IMPLIED, INCLUDING BUT NOT LIMITED TO THE WARRANTIES OF MERCHANTABILITY,
	FITNESS FOR A PARTICULAR PURPOSE AND NONINFRINGEMENT. IN NO EVENT SHALL THE
	AUTHORS OR COPYRIGHT HOLDERS BE LIABLE FOR ANY CLAIM, DAMAGES OR OTHER
	LIABILITY, WHETHER IN AN ACTION OF CONTRACT, TORT OR OTHERWISE, ARISING FROM,
	OUT OF OR IN CONNECTION WITH THE SOFTWARE OR THE USE OR OTHER DEALINGS IN THE
	SOFTWARE.
*)

// Performs rotation and updates heights until tree is balanced.
METHOD PROTECTED Balance
VAR_INPUT
    pNode : POINTER TO T_AVL_Node;
END_VAR
VAR 
    Balance_Factor : T_Position;
END_VAR
WHILE pNode <> 0 DO
	THIS^.Update_Height(pNode);
	
	Balance_Factor := THIS^.Get_Balance(pNode);
	
	IF Balance_Factor < -1 THEN
		IF THIS^.Get_Balance(pNode^.pRight) > 0 THEN THIS^.Rotate_Right(pNode^.pRight); END_IF
		THIS^.Rotate_Left(pNode);
	ELSIF Balance_Factor > 1 THEN
		IF THIS^.Get_Balance(pNode^.pLeft) < 0 THEN THIS^.Rotate_Left(pNode^.pLeft); END_IF
		THIS^.Rotate_Right(pNode);
		END_IF
		
	pNode := pNode^.pParent;
	END_WHILE
END_METHOD

// Deletes the node and its tree/sub-trees.
{warning disable C0394}
METHOD PROTECTED Clear_Node
VAR_INPUT
	pRoot : POINTER TO T_AVL_Node;
END_VAR
VAR
	fbNode_Stack : FB_Stack;
	pTmp : POINTER TO T_AVL_Node;
END_VAR
IF pRoot = 0 THEN RETURN; END_IF

fbNode_Stack.Push(pRoot);

WHILE NOT fbNode_Stack._Empty DO
	fbNode_Stack.Get(pTmp);
	fbNode_Stack.Pop();
	
	IF pTmp^.pRight <> 0 THEN fbNode_Stack.Push(pTmp^.pRight); END_IF
	IF pTmp^.pLeft <> 0 THEN fbNode_Stack.Push(pTmp^.pLeft); END_IF
	
	THIS^.Delete_Node(pTmp);
	END_WHILE
END_METHOD

// Creates a new node in dynamic memory with a clone of the generic item as it data.
METHOD PROTECTED Create_Node : POINTER TO ST_AVL_NODE
VAR_INPUT
	Item : T_Generic;
END_VAR
VAR_OUTPUT
	bSuccess : BOOL;
	Error : T_Error;
END_VAR
Create_Node := __NEW(ST_AVL_NODE);

IF Create_Node = 0 THEN Error := GVL_Errors.ERR_MALLOC_FAILED; RETURN; END_IF

Create_Node^.Data := F_Clone_Generic(Item, bSuccess => bSuccess, Error => Error);

IF NOT bSuccess THEN __DELETE(Create_Node); RETURN; END_IF
END_METHOD

// Safety deletes node.
// If the node and/or it's value/data is in dynamic memory it/they will be deleted.
METHOD PROTECTED Delete_Node
VAR_INPUT
	pNode : REFERENCE TO POINTER TO T_AVL_Node;
END_VAR
IF (pNode = 0) THEN RETURN; END_IF 

F_Delete_Generic(pNode^.Data);

CASE Tc2_System.F_CheckMemoryArea(pNode, 1) OF
	Tc2_System.E_TcMemoryArea.Dynamic: __DELETE(pNode);
ELSE
	pNode := 0;
	END_CASE
END_METHOD

// Finds the node with the smallest item in a tree or sub-tree.
METHOD PROTECTED Find_Minimum_Node : POINTER TO T_AVL_Node
VAR_INPUT
	pNode : POINTER TO T_AVL_Node;
END_VAR
IF pNode = 0 THEN RETURN; END_IF

WHILE pNode^.pLeft <> 0 DO
	pNode := pNode^.pLeft;
	END_WHILE
	
Find_Minimum_Node := pNode;
END_METHOD

// Gets the difference between the left and right sub-trees.
METHOD PROTECTED Get_Balance : T_Position
VAR_INPUT
	pNode : POINTER TO T_AVL_Node;
END_VAR
Get_Balance :=  THIS^.Get_Height(pNode^.pLeft) - THIS^.Get_Height(pNode^.pRight);
END_METHOD

// Safely gets the height of a sub-tree.
METHOD PROTECTED Get_Height : T_Position
VAR_INPUT
	pNode : POINTER TO T_AVL_Node;
END_VAR
Get_Height := SEL(pNode <> 0, -1, pNode^.Height);
END_METHOD

// Moves from node at source into the position of the destination.
METHOD PROTECTED Move_Node
VAR_INPUT
	pDestination, pSource : POINTER TO T_AVL_Node;
END_VAR
IF pDestination = 0 OR_ELSE pSource = 0 THEN RETURN; END_IF 

IF pDestination^.pParent = 0 THEN
	THIS^.pRoot := pSource;
ELSIF pDestination = pDestination^.pParent^.pLeft THEN
	pDestination^.pParent^.pLeft := pSource;
ELSE
	pDestination^.pParent^.pRight := pSource;
	END_IF
	
IF pSource <> 0 THEN
	pSource^.pParent := pDestination^.pParent;
	END_IF
END_METHOD

// Finds and removes a node from a tree/sub-tree and returns the new root of the tree/subtree.
METHOD PROTECTED Remove_Node : POINTER TO T_AVL_Node
VAR_INPUT
	pNode : REFERENCE TO POINTER TO T_AVL_Node;
END_VAR
VAR
	pSuccessor : POINTER TO T_AVL_Node;
END_VAR
IF (NOT __ISVALIDREF(pNode)) OR_ELSE pNode = 0 THEN RETURN; END_IF 

IF pNode^.pLeft = 0 THEN
	THIS^.Move_Node(pNode, pNode^.pRight);
	Remove_Node := pNode^.pRight;
ELSIF pNode^.pRight = 0 THEN 
	THIS^.Move_Node(pNode, pNode^.pLeft);
	Remove_Node := pNode^.pLeft;
ELSE
	Remove_Node := pSuccessor := THIS^.Find_Minimum_Node(pNode^.pRight);
	IF pSuccessor^.pParent <> pNode THEN 
		THIS^.Move_Node(pSuccessor, pSuccessor^.pRight);
		pSuccessor^.pRight := pNode^.pRight;
		pSuccessor^.pRight^.pParent := pSuccessor;
		END_IF
	THIS^.Move_Node(pNode, pSuccessor);
	pSuccessor^.pLeft := pNode^.pLeft;
	pSuccessor^.pLeft^.pParent := pSuccessor;
	END_IF

THIS^.Delete_Node(pNode);
END_METHOD

// Rotates a tree/sub-tree left.
METHOD PROTECTED Rotate_Left
VAR_INPUT
    pX : POINTER TO T_AVL_Node;
END_VAR
VAR
    pY : POINTER TO T_AVL_Node := pX^.pRight;
END_VAR
IF pY <> 0 THEN
	pX^.pRight := pY^.pLeft;
	IF pY^.pLeft <> 0 THEN pY^.pLeft^.pParent := pX; END_IF
	pY^.pParent := pX^.pParent;
	END_IF
	
IF pX^.pParent = 0 THEN
	THIS^.pRoot := pY;
ELSIF pX = pX^.pParent^.pLeft THEN
	pX^.pParent^.pLeft := pY;
ELSE
	pX^.pParent^.pRight := pY;
	END_IF
	
IF pY <> 0 THEN pY^.pLeft := pX; END_IF
	
pX^.pParent := pY;
THIS^.Update_Height(pX);
THIS^.Update_Height(pY);
END_METHOD

// Rotates a tree/sub-tree right.
METHOD PROTECTED Rotate_Right
VAR_INPUT
    pX : POINTER TO T_AVL_Node;
END_VAR
VAR
    pY : POINTER TO T_AVL_Node := pX^.pLeft;
END_VAR
IF pY <> 0 THEN
	pX^.pLeft := pY^.pRight;
	IF pY^.pRight <> 0 THEN pY^.pRight^.pParent := pX; END_IF
	pY^.pParent := pX^.pParent;
	END_IF
	
IF pX^.pParent = 0 THEN
	THIS^.pRoot := pY;
ELSIF pX = pX^.pParent^.pLeft THEN
	pX^.pParent^.pLeft := pY;
ELSE
	pX^.pParent^.pRight := pY;
	END_IF
	
IF pY <> 0 THEN pY^.pRight := pX; END_IF
	
pX^.pParent := pY;
THIS^.Update_Height(pX);
THIS^.Update_Height(pY);
END_METHOD

// Checks if an item is in a tree/ sub-tree.
METHOD PROTECTED Search_Node : POINTER TO T_AVL_Node
VAR_INPUT
	pNode : POINTER TO T_AVL_Node;
	Item : T_Generic;
END_VAR
WHILE pNode <> 0 DO
	CASE F_Compare_Generics(Item, pNode^.Data) OF
		T_Comparison.Less	: pNode := pNode^.pLeft;
		T_Comparison.Greater: pNode := pNode^.pRight; 
		T_Comparison.Equal	: 
			Search_Node := pNode;
			RETURN;
		END_CASE
	END_WHILE
END_METHOD

METHOD PROTECTED Update_Height
VAR_INPUT
	pNode : POINTER TO T_AVL_Node;
END_VAR
IF pNode = 0 THEN RETURN; END_IF
pNode^.Height := 1 + MAX(THIS^.Get_Height(pNode^.pLeft), THIS^.Get_Height(pNode^.pRight));
END_METHOD

// Traversal method for retrieving values in the tree set.
PROPERTY _Traversal : T_BST_Traversal
GET
_Traversal := THIS^.Traversal;
END_GET
SET
THIS^.Traversal := _Traversal;
END_SET
END_PROPERTY

// Empties/Clears/Deletes every item in the set.
METHOD Clear : I_Set
Clear := THIS^;

THIS^.Clear_Node(THIS^.pRoot);

IF THIS^.pValues <> 0 THEN
	THIS^.fbImmutable_Values_List(ipList := 0);
	__DELETE(THIS^.pValues);
	END_IF

THIS^.pRoot := 0;
THIS^._Count := 0;
END_METHOD

// Checks if item is contained in set.
METHOD Contains : BOOL
VAR_INPUT
	Item : ANY; // Item to find.
END_VAR
Contains := THIS^.Search_Node(THIS^.pRoot, Item) <> 0;
END_METHOD

{attribute 'hide'}
METHOD FB_exit : BOOL
VAR_INPUT
	bInCopyCode : BOOL; // if TRUE, the exit method is called for exiting an instance that is copied afterwards (online change).
END_VAR
// If this is an online change or this collection is empty then ignore. 
IF bInCopyCode THEN RETURN; END_IF

THIS^.Clear();
END_METHOD

// Gets an immutable list of the values in the set.
{warning disable C0394}
METHOD Get_Values : I_Immutable_List
VAR
	pCurrent, pPrevious, pTmp : POINTER TO T_AVL_Node := THIS^.pRoot;
	fbNode_Buffer : FB_Queue;
	bSuccess : BOOL;
END_VAR
IF THIS^.pValues = 0 THEN THIS^.pValues := __NEW(FB_Array_List(Initial_Capacity := 0)); END_IF
THIS^.fbImmutable_Values_List(ipList := THIS^.pValues^);
Get_Values := THIS^.fbImmutable_Values_List;

THIS^.pValues^.Clear();

IF pCurrent = 0 THEN RETURN; END_IF

WHILE (NOT fbNode_Buffer._Empty) OR_ELSE pCurrent <> 0 DO
	
	CASE THIS^._Traversal OF
		T_BST_Traversal.In_Order:
			IF pCurrent <> 0 THEN 
				fbNode_Buffer.Enqueue_At_Front(pCurrent);
				pCurrent := pCurrent^.pLeft;
			ELSE
				fbNode_Buffer.Get(pCurrent).Dequeue();
				THIS^.pValues^.Insert_Generic(THIS^.pValues^._Count, pCurrent^.Data);
				pCurrent := pCurrent^.pRight;
				END_IF
				
		T_BST_Traversal.Pre_Order:
			IF pCurrent <> 0 THEN 
				THIS^.pValues^.Insert_Generic(THIS^.pValues^._Count, pCurrent^.Data);
				IF pCurrent^.pRight <> 0 THEN fbNode_Buffer.Enqueue_At_Front(pCurrent^.pRight); END_IF
				pCurrent := pCurrent^.pLeft;
			ELSE
				fbNode_Buffer.Get(pCurrent).Dequeue();
				END_IF
			
		T_BST_Traversal.Post_Order:
			WHILE pCurrent <> 0 DO 
				fbNode_Buffer.Enqueue_At_Front(pCurrent);
				pCurrent := pCurrent^.pLeft;
				END_WHILE
				
			IF NOT fbNode_Buffer._Empty THEN
				fbNode_Buffer.Get(pTmp);
				pTmp := pTmp^.pRight;
				IF pTmp = 0 OR_ELSE pTmp = pPrevious THEN 
					fbNode_Buffer.Get(pCurrent).Dequeue();
					THIS^.pValues^.Insert_Generic(THIS^.pValues^._Count, pCurrent^.Data);
					pPrevious := pCurrent;
					pCurrent := 0;
				ELSE
					pCurrent := pTmp;
					END_IF
				END_IF
			
		T_BST_Traversal.Level_Order:
			THIS^.pValues^.Insert_Generic(THIS^.pValues^._Count, pCurrent^.Data);
			IF pCurrent^.pLeft <> 0 THEN fbNode_Buffer.Enqueue(pCurrent^.pLeft); END_IF
			IF pCurrent^.pRight <> 0 THEN fbNode_Buffer.Enqueue(pCurrent^.pRight); END_IF
			fbNode_Buffer.Get(pCurrent).Dequeue(bSuccess => bSuccess);
			IF NOT bSuccess THEN pCurrent := 0; END_IF
	ELSE
		RETURN;
		END_CASE
	END_WHILE
END_METHOD

// Insert item into set.
METHOD Insert 	: I_Set
VAR_INPUT
	Item : ANY; // Data to insert
END_VAR
VAR_OUTPUT
	bSuccess : BOOL; // Indicates whether operation was successful. Success = TRUE, Failure = FALSE
END_VAR
Insert := THIS^.Insert_Generic(Item, bSuccess => bSuccess);
END_METHOD

// Adds new generic item at into set.
// The set will store a copy of the generic item so as to not modify the original value outside it's scope.
METHOD Insert_Generic : I_Set
VAR_INPUT
	Item : T_Generic; // Item to store
END_VAR
VAR_OUTPUT
	bSuccess : BOOL; // Indicates whether operation was successful. Success = TRUE, Failure = FALSE
END_VAR
VAR
	pCurrent, pPrevious : POINTER TO T_AVL_Node;
END_VAR
Insert_Generic := THIS^;

pCurrent := THIS^.pRoot;
pPrevious := pCurrent;

WHILE pCurrent <> 0 DO
	pPrevious := pCurrent;
	CASE F_Compare_Generics(Item, pCurrent^.Data) OF
		T_Comparison.Less 	 : pCurrent := pCurrent^.pLeft;
		T_Comparison.Greater : pCurrent := pCurrent^.pRight;
		T_Comparison.Equal 	 : RETURN;
	ELSE
		THIS^._Error_Status := GVL_Errors.ERR_INVALID_COMPARISON;
		RETURN;
		END_CASE
	END_WHILE

pCurrent := THIS^.Create_Node(Item, bSuccess => bSuccess, Error => THIS^.Error);

IF NOT bSuccess THEN RETURN; END_IF

IF pPrevious = 0 THEN
	THIS^.pRoot := pCurrent;
ELSE
	CASE F_Compare_Generics(Item, pPrevious^.Data) OF
		T_Comparison.Less: pPrevious^.pLeft := pCurrent;
	ELSE
		pPrevious^.pRight := pCurrent;
		END_CASE
	END_IF

pCurrent^.pParent := pPrevious;
	
THIS^.Balance(pCurrent);
THIS^.Increment_Count();
END_METHOD

// Removes item from the set.
METHOD Remove : I_Set
VAR_INPUT
	Item : ANY; // Data to remove
END_VAR
VAR_OUTPUT
	bSuccess : BOOL; // Indicates whether operation was successful. Success = TRUE, Failure = FALSE
END_VAR
Remove := THIS^.Remove_Generic(Item, bSuccess => bSuccess);
END_METHOD

// Removes generic item from the set.
METHOD Remove_Generic : I_Set
VAR_INPUT
	Item : T_Generic; // Data to remove
END_VAR
VAR_OUTPUT
	bSuccess : BOOL; // Indicates whether operation was successful. Success = TRUE, Failure = FALSE
END_VAR
VAR
	pTmp : POINTER TO T_AVL_Node;
END_VAR
Remove_Generic := THIS^;

pTmp := THIS^.Search_Node(THIS^.pRoot, Item);

IF pTmp = 0 THEN RETURN; END_IF

THIS^.Balance(THIS^.Remove_Node(pTmp));

THIS^.Decrement_Count();
THIS^.Clear_Error();

IF THIS^._Empty THEN THIS^.pRoot := 0; END_IF

bSuccess := TRUE;
END_METHOD

END_FUNCTION_BLOCK

// POUs/Function Blocks/Enumerators/FB_Enumerator
// Base function block for enumerators.
{attribute 'enable_dynamic_creation'}
{attribute 'no_explicit_call' := 'direct call for this function block is not allowed'}
FUNCTION_BLOCK INTERNAL ABSTRACT FB_Enumerator IMPLEMENTS I_Enumerator
VAR
	ipEnumerator : REFERENCE TO I_Enumerator;
	Index : T_Position := -1;
END_VAR

// Gets an item in the collection at current positon of the enumerator.
METHOD ABSTRACT Current : I_Enumerator
VAR_INPUT
	Item : ANY;
END_VAR
END_METHOD

// Gets an item in the collection at current positon of the enumerator as a string.
METHOD ABSTRACT Current_As_String : I_Enumerable
VAR_INPUT
	sItem : REFERENCE TO STRING;
END_VAR
END_METHOD

// Releases resources allocated to the enumerator. Returns TRUE if successful.
METHOD FINAL Dispose : BOOL
IF __ISVALIDREF(THIS^.ipEnumerator) THEN RETURN; END_IF
THIS^.ipEnumerator := 0;
__DELETE(THIS);
END_METHOD

{attribute 'hide'}
METHOD ABSTRACT FB_exit : BOOL
VAR_INPUT
	bInCopyCode : BOOL; // if TRUE, the exit method is called for exiting an instance that is copied afterwards (online change).
END_VAR
END_METHOD

{attribute 'hide'}
METHOD FB_init : BOOL
VAR_INPUT
	bInitRetains : BOOL; // if TRUE, the retain variables are initialized (warm start / cold start)
	bInCopyCode : BOOL;  // if TRUE, the instance afterwards gets moved into the copy code (online change)
	ipEnumerator : REFERENCE TO I_Enumerator;
END_VAR
IF bInCopyCode OR_ELSE NOT __ISVALIDREF(ipEnumerator) THEN RETURN; END_IF
IF ipEnumerator <> 0 THEN ipEnumerator.Dispose(); END_IF
THIS^.ipEnumerator REF= ipEnumerator;
END_METHOD

// Advances the enumerator to the next item of the collection.
METHOD ABSTRACT Next : BOOL
END_METHOD

// Sets the enumerator to its initial position, which is before the first element in the collection.
METHOD ABSTRACT Reset : I_Enumerator
END_METHOD

END_FUNCTION_BLOCK

// POUs/Function Blocks/Misc/FB_Free
// Frees pointer when this instance of the FB leaves the scope;
{attribute 'no_explicit_call' := 'direct call for this function block is not allowed'}
FUNCTION_BLOCK INTERNAL FINAL FB_Free
VAR
	_pValue : REFERENCE TO POINTER TO BYTE;
END_VAR

{attribute 'hide'} 
METHOD FB_exit : BOOL
VAR_INPUT
	bInCopyCode : BOOL; // if TRUE, the exit method is called for exiting an instance that is copied afterwards (online change).
END_VAR
IF bInCopyCode THEN RETURN; END_IF
IF NOT __ISVALIDREF(THIS^._pValue) THEN RETURN; END_IF
IF THIS^._pValue <> 0 THEN __DELETE(THIS^._pValue); END_IF
END_METHOD

{attribute 'hide'} 
{attribute 'no_explicit_call' := 'do not call this POU directly'}
METHOD FB_init : BOOL
VAR_INPUT
	bInitRetains 	: BOOL; // if TRUE, the retain variables are initialized (warm start / cold start)
	bInCopyCode 	: BOOL;  // if TRUE, the instance afterwards gets moved into the copy code (online change)
	pValue 			: REFERENCE TO POINTER TO BYTE; // Pointer to be freed on exit
END_VAR
THIS^._pValue REF= pValue;
END_METHOD

END_FUNCTION_BLOCK

// POUs/Functions/F_Any_To_Generic
FUNCTION F_Any_To_Generic : T_Generic
VAR_INPUT
	Value : ANY;
END_VAR

F_Any_To_Generic := Value;

END_FUNCTION

// POUs/Functions/F_Compare_Any
// Compares value A to generic value B of any type and returns the evaluation.
FUNCTION F_Compare_Any : T_Comparison
VAR_INPUT
	A : ANY;
	B : ANY;
END_VAR

F_Compare_Any := F_Compare_Generics(A, B);

END_FUNCTION

// POUs/Functions/F_String_Convertable_Generic
// Checks if value can be converted to string
FUNCTION F_String_Convertable_Generic : BOOL
VAR_INPUT
	Value : T_Generic;
END_VAR

CASE Value.TypeClass OF
	__SYSTEM.TYPE_CLASS.TYPE_STRING,
	__SYSTEM.TYPE_CLASS.TYPE_WSTRING,
	__SYSTEM.TYPE_CLASS.TYPE_BOOL,
	__SYSTEM.TYPE_CLASS.TYPE_BYTE,
	__SYSTEM.TYPE_CLASS.TYPE_WORD,
	__SYSTEM.TYPE_CLASS.TYPE_DWORD,
	__SYSTEM.TYPE_CLASS.TYPE_LWORD,
	__SYSTEM.TYPE_CLASS.TYPE_SINT,
	__SYSTEM.TYPE_CLASS.TYPE_INT,
	__SYSTEM.TYPE_CLASS.TYPE_DINT,
	__SYSTEM.TYPE_CLASS.TYPE_LINT,
	__SYSTEM.TYPE_CLASS.TYPE_USINT,
	__SYSTEM.TYPE_CLASS.TYPE_UINT,
	__SYSTEM.TYPE_CLASS.TYPE_UDINT,
	__SYSTEM.TYPE_CLASS.TYPE_ULINT,
	__SYSTEM.TYPE_CLASS.TYPE_REAL,
	__SYSTEM.TYPE_CLASS.TYPE_LREAL,
	__SYSTEM.TYPE_CLASS.TYPE_TIME,
	__SYSTEM.TYPE_CLASS.TYPE_LTIME,
	__SYSTEM.TYPE_CLASS.TYPE_DATE,
	__SYSTEM.TYPE_CLASS.TYPE_DATEANDTIME,
	__SYSTEM.TYPE_CLASS.TYPE_TIMEOFDAY,
	__SYSTEM.TYPE_CLASS.TYPE_POINTER:
		F_String_Convertable_Generic := TRUE;
ELSE
	RETURN;
END_CASE

END_FUNCTION

// POUs/Functions/F_String_To_Any
// Converts string to generic.
FUNCTION F_String_To_Any
VAR_INPUT
	sValue : REFERENCE TO STRING;
	Value : ANY;
END_VAR
VAR_OUTPUT
	bSuccess : BOOL;
	Error : T_Error := GVL_Errors.ERR_NO_ERROR;
END_VAR
VAR
	pBool			: POINTER TO BOOL;
    pByte			: POINTER TO BYTE;
    pWord			: POINTER TO WORD;
    pDWord			: POINTER TO DWORD;
    pLWord			: POINTER TO LWORD;
    pSint			: POINTER TO SINT;
    pInt			: POINTER TO INT;
    pDint			: POINTER TO DINT;
    pLint			: POINTER TO LINT;
    pUSint			: POINTER TO USINT;
    pUInt			: POINTER TO UINT;
    pUDint			: POINTER TO UDINT;
    pULint			: POINTER TO ULINT;
    pReal			: POINTER TO REAL;
    pLReal			: POINTER TO LREAL;
    pString			: POINTER TO STRING(255);
    pWString		: POINTER TO WSTRING;
    pTime			: POINTER TO TIME;
    pDate			: POINTER TO DATE;
    pDate_And_Time	: POINTER TO DATE_AND_TIME;
    pTime_Of_Day	: POINTER TO TIME_OF_DAY;
    pPointer		: POINTER TO PVOID;
	pLTime 			: POINTER TO LTIME;
END_VAR

IF (Value.pValue = 0) OR_ELSE (NOT __ISVALIDREF(sValue)) THEN 
	Error := GVL_Errors.ERR_INVALID_REFERENCE;
	RETURN; 
	END_IF;

IF NOT F_String_Convertable_Generic(Value) THEN
	Error := GVL_Errors.ERR_INVALID_CONVERSION;
	RETURN;
	END_IF

CASE Value.TypeClass OF 
	__SYSTEM.TYPE_CLASS.TYPE_BOOL:
		pBool := Value.pValue;
		pBool^ := TO_BOOL(sValue);
		
    __SYSTEM.TYPE_CLASS.TYPE_BYTE:
		pByte := Value.pValue;
		pByte^ := TO_BYTE(sValue);
		
    __SYSTEM.TYPE_CLASS.TYPE_WORD:
		pWord := Value.pValue;
		pWord^ := TO_WORD(sValue);
		
    __SYSTEM.TYPE_CLASS.TYPE_DWORD:
		pDWord := Value.pValue;
		pDWord^ := TO_DWORD(sValue);
		
    __SYSTEM.TYPE_CLASS.TYPE_LWORD:
		pLWord := Value.pValue;
		pLWord^ := TO_LWORD(sValue);
		
    __SYSTEM.TYPE_CLASS.TYPE_SINT:
		pSint := Value.pValue;
		pSint^ := TO_SINT(sValue);
		
    __SYSTEM.TYPE_CLASS.TYPE_INT:
		pInt := Value.pValue;
		pInt^ := TO_INT(sValue);
		
    __SYSTEM.TYPE_CLASS.TYPE_DINT:
		pDint := Value.pValue;
		pDint^ := TO_DINT(sValue);
		
    __SYSTEM.TYPE_CLASS.TYPE_LINT:
		pLint := Value.pValue;
		pLint^ := TO_LINT(sValue);
		
    __SYSTEM.TYPE_CLASS.TYPE_USINT:
		pUSint := Value.pValue;
		pUSint^ := TO_USINT(sValue);
		
    __SYSTEM.TYPE_CLASS.TYPE_UINT:
		pUInt := Value.pValue;
		pUInt^ := TO_UINT(sValue);
		
    __SYSTEM.TYPE_CLASS.TYPE_UDINT:
		pUDint := Value.pValue;
		pUDint^ := TO_UDINT(sValue);
		
    __SYSTEM.TYPE_CLASS.TYPE_ULINT:
		pULint := Value.pValue;
		pULint^ := TO_ULINT(sValue);
		
   __SYSTEM.TYPE_CLASS.TYPE_REAL:
		pReal := Value.pValue;
		pReal^ := TO_REAL(sValue);
		
    __SYSTEM.TYPE_CLASS.TYPE_LREAL:
		pLReal := Value.pValue;
		pLReal^ := TO_LREAL(sValue);
		
    __SYSTEM.TYPE_CLASS.TYPE_STRING:
		Tc2_Utilities.STRNCPY(Value.pValue, ADR(sValue), TO_UDINT(Value.diSize)); 
		
   __SYSTEM.TYPE_CLASS.TYPE_WSTRING:
   		Tc2_Utilities.STRING_TO_WSTRING2(Value.pValue, ADR(sValue), TO_UDINT(Value.diSize));
		
    __SYSTEM.TYPE_CLASS.TYPE_TIME:
		pTime := Value.pValue;
		pTime^ := TO_TIME(sValue);
		
	__SYSTEM.TYPE_CLASS.TYPE_LTIME:
		pLTime := Value.pValue;
		pLTime^ := TO_LTIME(sValue);
		
    __SYSTEM.TYPE_CLASS.TYPE_DATE:
		pDate := Value.pValue;
		pDate^ := TO_DATE(sValue);
		
    __SYSTEM.TYPE_CLASS.TYPE_DATEANDTIME:
		pDate_And_Time := Value.pValue;
		pDate_And_Time^ := TO_DT(sValue);
		
    __SYSTEM.TYPE_CLASS.TYPE_TIMEOFDAY:
		pTime_Of_Day := Value.pValue;
		pTime_Of_Day^ := TO_TOD(sValue);
	
	__SYSTEM.TYPE_CLASS.TYPE_POINTER:
		pPointer := Value.pValue;
		pPointer^ := Tc2_Utilities.STRING_TO_PVOID(sValue);
END_CASE

bSuccess := TRUE;

END_FUNCTION

// POUs/MAIN
PROGRAM INTERNAL MAIN
VAR
	Data : ARRAY[0..10] OF DINT := [1,2,3,4,5,6,7,8,9,10];
	rData: ARRAY[0..10] OF DINT;
	Size : UDINT;
	i,j : T_Position;
	ipImm : I_Immutable_List;
	bAdd, bRemove, bClear : BOOL;
	fbArray : FB_Array(10);
	fbImm_Arr : FB_Immutable_Array;
	fbImm_Map : FB_Immutable_Map;
	fbImm_Set : FB_Immutable_Set;
	fbArray_List : FB_Array_List(0);
	fbList : FB_List;
	fbQueue : FB_Queue;
	fbStack : FB_Stack;
	fbDeque : FB_Deque;
	fbTree_Set : FB_Tree_Set;
	fbHash_Set : FB_Hash_Set(3);
	fbTree_Map : FB_Tree_Map;
	fbHash_Map : FB_Hash_Map(3);
	fbMultiset : FB_Tree_Multiset;
END_VAR

Size := SIZEOF(fbHash_Set);

IF bAdd THEN
	bAdd := FALSE;
	END_IF

IF bRemove THEN
	bRemove := FALSE;
	END_IF
	
IF bClear THEN
	bClear := FALSE;
	END_IF

END_PROGRAM

// Project Information/F_GetCompany
// This function has been automatically generated from the project information.
{attribute 'signature_flag' := '1073741824'}
{attribute 'TcGenerated'}
{attribute 'no-analysis'}
FUNCTION F_GetCompany : WSTRING
VAR_INPUT
	
END_VAR

F_GetCompany := "FisoThemes";

END_FUNCTION

// Project Information/F_GetTitle
// This function has been automatically generated from the project information.
{attribute 'signature_flag' := '1073741824'}
{attribute 'TcGenerated'}
{attribute 'no-analysis'}
FUNCTION F_GetTitle : WSTRING
VAR_INPUT
	
END_VAR

F_GetTitle := "TwinCat Dynamic Collections";

END_FUNCTION

// Project Information/F_GetVersion
// This function has been automatically generated from the project information.
{attribute 'signature_flag' := '1073741824'}
{attribute 'TcGenerated'}
{attribute 'no-analysis'}
FUNCTION F_GetVersion : ST_LibVersion
VAR_INPUT
	
END_VAR

F_GetVersion.iMajor := 1;
F_GetVersion.iMinor := 0;
F_GetVersion.iBuild := 5;
F_GetVersion.iRevision := 28;

END_FUNCTION
